// TwinCAT 3 PLC project Universalsteuerung_0663
// ProgramVersion: 3.1.4026.13
// libraries:
//   QSC_Einzelschritte, * (Q+S Control AG)
//   Tc2_MC2, * (Beckhoff Automation GmbH)
//   Tc2_Standard, * (Beckhoff Automation GmbH)
//   Tc2_SUPS, * (Beckhoff Automation GmbH)
//   Tc2_System, * (Beckhoff Automation GmbH)
//   Tc2_Utilities, * (Beckhoff Automation GmbH)
//   Tc3_EventLogger, * (Beckhoff Automation GmbH)
//   Tc3_IotBase, * (Beckhoff Automation GmbH)
//   Tc3_JsonXml, * (Beckhoff Automation GmbH)
//   Tc3_Module, * (Beckhoff Automation GmbH)
//   VisuDialogs, * (System)
//   VisuSymbols,3.5.10.0,System
// project tree:
//   DUTs/Enums/ AblaufStatus.TcDUT, AktorStatus.TcDUT, Artikeltyp.TcDUT, InitStatus.TcDUT, ResetStatus.TcDUT, StatusbarFarbe.TcDUT, StatusGreifer.TcDUT, StatusZufuehrung.TcDUT, Wartungen.TcDUT
//   DUTs/Enums/Apromace/ Antwort.TcDUT, AuftragsStatus.TcDUT, MessageArt.TcDUT
//   DUTs/Structs/EL9227_Überstromschutzklemme/ ST_BIT2.TcDUT, ST_Control.TcDUT, ST_EL9227_IN.TcDUT, ST_Status.TcDUT
//   DUTs/Structs/ ST_Ablauf_Konfig.TcDUT, ST_ArtikelParameter.TcDUT, ST_AufnahmeInfo.TcDUT, ST_EventTabelle.TcDUT, ST_Programme.TcDUT, ST_Aktor_Konfig.TcDUT, ST_QrCode.TcDUT, ST_Reihenfolge.TcDUT, ST_SchrittQueue.TcDUT, ST_Station.TcDUT, ST_Stueckzaehler.TcDUT, ST_UeberstromTabelle.TcDUT, ST_Wartung.TcDUT
//   / GlobalTextList.TcGTLO, PlcTask.TcTTO, VisualizationManager.TcVMO (not stored), VISU_TASK.TcTTO
//   GVLs/ ArtikelParam.TcGVL, Exc.TcGVL, Parameter.TcGVL
//   POUs/EventLogger/ EventLogger.TcPOU, FB_Arguments.TcPOU, FB_Event.TcPOU
//   POUs/ FB_Aktor.TcPOU, FB_Datei.TcPOU, FB_EL9227.TcPOU, FB_Handheld.TcPOU, FB_Hmi.TcPOU, FB_Output.TcPOU, FB_Schrittbetrieb.TcPOU, FB_Station01.TcPOU, FB_Stundenleistung.TcPOU, FB_Turmleuchte.TcPOU, FB_Wartung.TcPOU, FB_Zykluszeit.TcPOU, MAIN.TcPOU, Tools.TcPOU
//   POUs/Interfaces/ IF_Station.TcIO, IF_TeilBereitstellen.TcIO, IF_TeilHolen.TcIO
//   POUs/StdStationen/ FB_Station.TcPOU, FB_StationMitZuf.TcPOU, FB_StationMitZufUndVer.TcPOU
//   VISUs/ Konfig2.TcVIS, TL_Aktoren.TcTLO, Diagnose.TcVIS, EventLogger.TcVIS, TL_JaNein.TcTLO, Wartung.TcVIS, Handbetrieb.TcVIS, Konfig1.TcVIS, ImagePool.TcIPO (not stored), Zyklusbetrieb.TcVIS
// real-time tasks:
//   TASK PlcTask: cycle T#10ms, priority 20, ADS port 350
//   TASK VISU_TASK: cycle T#50000us, priority 30, ADS port 351
// I/O:
//   DEVICE Device 1 (EtherCAT), AmsNetId 10.200.30.201.2.1
//     601A1 (EK1100) [EK1100 EtherCAT Coupler (2A E-Bus)]
//       601A2 (EL9227-5500) [EL9227-5500 Overcurrent protection 24V DC, 2Ch., max. 10A (sum), adjustable, extended functionalities]
//       601A3 (EL2911) [EL2911, Potential supply terminal (10 A) with 4 Ch. Safety Inputs, TwinSAFE]
//         modules: Module 2 (FSOUT), Module 3 (DEVICEIO), Module 4 (FSLOGIC)
//       601A5 (EL9227-5500) [EL9227-5500 Overcurrent protection 24V DC, 2Ch., max. 10A (sum), adjustable, extended functionalities]
//       602A1(EL1008) [EL1008 8Ch. Dig. Input 24V, 3ms]
//       602A2 (EL2008-0015) [EL2008-0015 8Ch. Dig. Output 24V DC, 0.35A, not short-circuit proof]
//       602A4 (EL9184) [EL9184 Potential Connection, 8 x 24V, 8 x Ground]
//       (EL9011) [EL9011 End Terminal]
//     Box 15 (EP2339-0003) [EP2339-0003 16 Ch. Dig. Input/Output 24V, 0,5A, 10-Pole Plug Connector]
//     Box 16 (CTEU-EtherCAT Modular) [CTEU-EtherCAT Fieldbus modular]
//       modules: Module 1 (VAEM-L1-S-8-PT [16DO])
// variable links:
//   Universalsteuerung_0663/Universalsteuerung_0663 Instance <-> Device 1 (EtherCAT)/601A1 (EK1100)/601A2 (EL9227-5500)
//     PlcTask Inputs/MAIN.fb601A2.stKanal[1].nCurrent <-> OCP Inputs Channel 1/Current
//     PlcTask Inputs/MAIN.fb601A2.stKanal[2].nCurrent <-> OCP Inputs Channel 2/Current
//     PlcTask Inputs/MAIN.fb601A2.stKanal[1].nLoad <-> OCP Inputs Channel 1/Load
//     PlcTask Inputs/MAIN.fb601A2.stKanal[2].nLoad <-> OCP Inputs Channel 2/Load
//     PlcTask Inputs/MAIN.fb601A2.stKanal[1].nVoltageIn <-> OCP Inputs Channel 1/Voltage In
//     PlcTask Inputs/MAIN.fb601A2.stKanal[2].nVoltageIn <-> OCP Inputs Channel 2/Voltage In
//     PlcTask Inputs/MAIN.fb601A2.stKanal[1].nVoltageOut <-> OCP Inputs Channel 1/Voltage Out
//     PlcTask Inputs/MAIN.fb601A2.stKanal[2].nVoltageOut <-> OCP Inputs Channel 2/Voltage Out
//     PlcTask Inputs/MAIN.fb601A2.stKanal[1].stStatus <-> OCP Inputs Channel 1/Status
//     PlcTask Inputs/MAIN.fb601A2.stKanal[2].stStatus <-> OCP Inputs Channel 2/Status
//     PlcTask Outputs/MAIN.fb601A2.stKanal[1].stControl <-> OCP Outputs Channel 1/Control
//     PlcTask Outputs/MAIN.fb601A2.stKanal[2].stControl <-> OCP Outputs Channel 2/Control
//   Universalsteuerung_0663/Universalsteuerung_0663 Instance <-> Device 1 (EtherCAT)/601A1 (EK1100)/601A3 (EL2911)
//     PlcTask Inputs/MAIN.bE_LampeNHReset <-> StandardInputs/TwinSafeGroup1.LampeNHResetOutSPS_14
//     PlcTask Inputs/MAIN.bE_LampeNotHalt <-> StandardInputs/TwinSafeGroup1.LampeNotHaltOutSPS_88
//     PlcTask Inputs/MAIN.bE_NotHalt <-> StandardInputs/TwinSafeGroup1.NotHaltOutSPS_19
//     PlcTask Inputs/MAIN.bE_SafetyComErr <-> StandardInputs/TwinSafeGroup1.ComError_16
//     PlcTask Inputs/MAIN.bE_SafetyInRun <-> StandardInputs/TwinSafeGroup1.SafetyInRun_86
//     PlcTask Inputs/MAIN.bE_SafetyOtherErr <-> StandardInputs/TwinSafeGroup1.OtherError_17
//     PlcTask Inputs/MAIN.bE_SafetyProgStop <-> StandardInputs/TwinSafeGroup1.ProgStop_64
//     PlcTask Outputs/MAIN.bA_Hauptventil <-> StandardOutputs/TwinSafeGroup1.HauptventilSPS_48
//     PlcTask Outputs/MAIN.bA_SafetyReset <-> StandardOutputs/TwinSafeGroup1.ErrorAcknowledgement_1
//     PlcTask Outputs/MAIN.bA_SafetyRun <-> StandardOutputs/TwinSafeGroup1.Run_47
//   Universalsteuerung_0663/Universalsteuerung_0663 Instance <-> Device 1 (EtherCAT)/601A1 (EK1100)/601A5 (EL9227-5500)
//     PlcTask Inputs/MAIN.fb601A5.stKanal[1].nCurrent <-> OCP Inputs Channel 1/Current
//     PlcTask Inputs/MAIN.fb601A5.stKanal[2].nCurrent <-> OCP Inputs Channel 2/Current
//     PlcTask Inputs/MAIN.fb601A5.stKanal[1].nLoad <-> OCP Inputs Channel 1/Load
//     PlcTask Inputs/MAIN.fb601A5.stKanal[2].nLoad <-> OCP Inputs Channel 2/Load
//     PlcTask Inputs/MAIN.fb601A5.stKanal[1].nVoltageIn <-> OCP Inputs Channel 1/Voltage In
//     PlcTask Inputs/MAIN.fb601A5.stKanal[2].nVoltageIn <-> OCP Inputs Channel 2/Voltage In
//     PlcTask Inputs/MAIN.fb601A5.stKanal[1].nVoltageOut <-> OCP Inputs Channel 1/Voltage Out
//     PlcTask Inputs/MAIN.fb601A5.stKanal[2].nVoltageOut <-> OCP Inputs Channel 2/Voltage Out
//     PlcTask Inputs/MAIN.fb601A5.stKanal[1].stStatus <-> OCP Inputs Channel 1/Status
//     PlcTask Inputs/MAIN.fb601A5.stKanal[2].stStatus <-> OCP Inputs Channel 2/Status
//     PlcTask Outputs/MAIN.fb601A5.stKanal[1].stControl <-> OCP Outputs Channel 1/Control
//     PlcTask Outputs/MAIN.fb601A5.stKanal[2].stControl <-> OCP Outputs Channel 2/Control
//   Universalsteuerung_0663/Universalsteuerung_0663 Instance <-> Device 1 (EtherCAT)/601A1 (EK1100)/602A1(EL1008)
//     PlcTask Inputs/MAIN.bE_LuftdruckIO <-> Channel 5/Input
//     PlcTask Inputs/MAIN.bE_Taste_Schritt <-> Channel 4/Input
//     PlcTask Inputs/MAIN.bE_Taste_Start <-> Channel 1/Input
//     PlcTask Inputs/MAIN.bE_Taste_Stoerung <-> Channel 3/Input
//     PlcTask Inputs/MAIN.bE_Taste_Stop <-> Channel 2/Input
//   Universalsteuerung_0663/Universalsteuerung_0663 Instance <-> Device 1 (EtherCAT)/601A1 (EK1100)/602A2 (EL2008-0015)
//     PlcTask Outputs/MAIN.bA_Lampe_NHReset <-> Channel 4/Output
//     PlcTask Outputs/MAIN.bA_Lampe_NotHalt <-> Channel 5/Output
//     PlcTask Outputs/MAIN.bA_Lampe_Schritt <-> Channel 6/Output
//     PlcTask Outputs/MAIN.bA_Lampe_Start <-> Channel 1/Output
//     PlcTask Outputs/MAIN.bA_Lampe_Stoerung <-> Channel 3/Output
//     PlcTask Outputs/MAIN.bA_Lampe_Stop <-> Channel 2/Output
//   Universalsteuerung_0663/Universalsteuerung_0663 Instance <-> Device 1 (EtherCAT)/Box 15 (EP2339-0003)
//     PlcTask Inputs/MAIN.bE_Fussschalter <-> DI Inputs Channel 2/Input 1
//     PlcTask Inputs/MAIN.fbSt1.bE_Sensor[{1..8}] <-> DI Inputs Channel 1/Input {1..8}  (8 links)
//     PlcTask Outputs/MAIN.fbSt1.bA_extGeraetStart <-> DO Outputs Channel 2/Output 2
//   Universalsteuerung_0663/Universalsteuerung_0663 Instance <-> Device 1 (EtherCAT)/Box 16 (CTEU-EtherCAT Modular)
//     PlcTask Outputs/MAIN.fbSt1.fbAktor[1].bA_arbeitsPos <-> Module 1 (VAEM-L1-S-8-PT [16DO])/Outputs/C1 Output[0]
//     PlcTask Outputs/MAIN.fbSt1.fbAktor[2].bA_arbeitsPos <-> Module 1 (VAEM-L1-S-8-PT [16DO])/Outputs/C1 Output[2]
//     PlcTask Outputs/MAIN.fbSt1.fbAktor[3].bA_arbeitsPos <-> Module 1 (VAEM-L1-S-8-PT [16DO])/Outputs/C1 Output[4]
//     PlcTask Outputs/MAIN.fbSt1.fbAktor[4].bA_arbeitsPos <-> Module 1 (VAEM-L1-S-8-PT [16DO])/Outputs/C1 Output[6]
//     PlcTask Outputs/MAIN.fbSt1.fbAktor[5].bA_arbeitsPos <-> Module 1 (VAEM-L1-S-8-PT [16DO])/Outputs/C2 Output[0]
//     PlcTask Outputs/MAIN.fbSt1.fbAktor[6].bA_arbeitsPos <-> Module 1 (VAEM-L1-S-8-PT [16DO])/Outputs/C2 Output[2]

CONFIGURATION Universalsteuerung_0663
    RESOURCE PLC ON TwinCAT3
        TASK PlcTask(INTERVAL := T#10ms, PRIORITY := 20);
        TASK VISU_TASK(INTERVAL := T#50000us, PRIORITY := 30);
        PROGRAM MAIN WITH PlcTask : MAIN;
        PROGRAM VisuElems_Visu_Prg WITH VISU_TASK : VisuElems.Visu_Prg;
    END_RESOURCE
END_CONFIGURATION

// ---- DUTs/Enums/AblaufStatus.TcDUT
{attribute 'qualified_only'}
//{attribute 'strict'}
{attribute 'to_string'}
TYPE AblaufStatus :
(
//	default				:= 0,
//	bereit				:= 1,
//	error				:= 2,
//	produziert			:= 3,
//	fertig				:= 5,
//	popUp				:= 6,
	
//	aktor01Vor			:= 10,
//	aktor01Zurueck		:= 11,
//	aktor02Vor			:= 20,
//	aktor02Zurueck		:= 21,
//	aktor03Vor			:= 30,
//	aktor03Zurueck		:= 31,
//	aktor04Vor			:= 40,
//	aktor04Zurueck		:= 41,
//	aktor05Vor			:= 50,
//	aktor05Zurueck		:= 51,
//	aktor06Vor			:= 60,
//	aktor06Zurueck		:= 61,
	
//	teilAnwesend		:= 80,
//	extGeraetBereit		:= 81,
//	extGeraetStart		:= 82,
//	warten				:= 90,
	
//	nameUeberpruefen 	:= 200,
//	freierPlatzsuchen 	:= 201,
//	programmSpeichern 	:= 202,
//	programmAnzeigen	:= 203,
//	programmLoeschen	:= 204

	default				:= 0,
	aktor01Vor			:= 1,
	aktor01Zurueck		:= 2,
	aktor02Vor			:= 3,
	aktor02Zurueck		:= 4,
	aktor03Vor			:= 5,
	aktor03Zurueck		:= 6,
	aktor04Vor			:= 7,
	aktor04Zurueck		:= 8,
	aktor05Vor			:= 9,
	aktor05Zurueck		:= 10,
	aktor06Vor			:= 11,
	aktor06Zurueck		:= 12,
	teilAnwesend		:= 13,
	extGeraetBereit		:= 14,
	extGeraetStart		:= 15,
	extGeraetFertig		:= 16,
	warten				:= 17,
	schritt				:= 18,
	
	bereit				:= 30,
	error				:= 31,
	produziert			:= 32,
	fertig				:= 33,
	popUp				:= 34,
	naechsterSchritt	:= 35,
	
	nameUeberpruefen 	:= 200,
	freierPlatzsuchen 	:= 201,
	programmSpeichern 	:= 202,
	programmAnzeigen	:= 203,
	programmLoeschen	:= 204,
	
	oeffnen				:= 300,
	wartenOffen			:= 301,
	schreiben			:= 302,
	wartenGeschrieben	:= 303,
	schliessen			:= 304,
	wartenGeschlossen	:= 305
	
	
	

	
);
END_TYPE

// ---- DUTs/Enums/AktorStatus.TcDUT
{attribute 'qualified_only'}
{attribute 'strict'}
{attribute 'to_string'}
TYPE AktorStatus :
(
	default := 0,
	inRP,
	inAP,
	
	zuRP,
	zuAP
);
END_TYPE

// ---- DUTs/Enums/Apromace/Antwort.TcDUT
{attribute 'qualified_only'}
{attribute 'strict'}
TYPE Antwort :
(
	pending,	//wartet auf Antwort
	timeout,
	ok,
	error,
	ignored,	//Ignore flag aktiviert
	expired		//Quittiert nach Error
);
END_TYPE

// ---- DUTs/Enums/Apromace/AuftragsStatus.TcDUT
{attribute 'qualified_only'}
{attribute 'strict'}
TYPE AuftragsStatus :
(
	scan,
	start,
	end,
	vorwahl
);
END_TYPE

// ---- DUTs/Enums/Apromace/MessageArt.TcDUT
{attribute 'qualified_only'}
{attribute 'strict'}
{attribute 'to_string'}
TYPE MessageArt :
(
	status,
	auftrag,
	daten,
	parameter
);
END_TYPE

// ---- DUTs/Enums/Artikeltyp.TcDUT
{attribute 'qualified_only'}
{attribute 'strict'}
{attribute 'to_string'}
TYPE Artikeltyp :
(
	default 				:= 0,
	br51,
	br84
);
END_TYPE

// ---- DUTs/Enums/InitStatus.TcDUT
{attribute 'qualified_only'}
{attribute 'strict'}
{attribute 'to_string'}
TYPE InitStatus :
(
	default := 0,
	bereit,
	steuerungEin,
	safety,
	resetSafety,
	luftdruck,
	fertig,
	stationen,
	aktor1,
	aktor2,
	aktor3,
	aktor4,
	aktor5,
	aktor6
);
END_TYPE

// ---- DUTs/Enums/ResetStatus.TcDUT
{attribute 'qualified_only'}
{attribute 'strict'}
{attribute 'to_string'}
TYPE ResetStatus :
(
	default := 0,
	bereit,
	ablaufAbbrechen,
	ausschalten,
	fertig,
	aktoren,
	kommunikationAbgebrochen
);
END_TYPE

// ---- DUTs/Enums/StatusbarFarbe.TcDUT
{attribute 'qualified_only'}
TYPE StatusbarFarbe :
(
	default := 0,
	rot :=1,
	orange := 2,
	gruen := 3,
	blau := 4
);
END_TYPE

// ---- DUTs/Enums/StatusGreifer.TcDUT
{attribute 'qualified_only'}
{attribute 'strict'}
{attribute 'to_string'}
TYPE StatusGreifer :
(
	default := 0,
	keinTeil,
	teilHolen,
	teilGeholt,
	teilEinlegen,
	teilEntnehmen,
	teilEntnommen,
	teilAblegen,
	teilAbgelegt,
	teilGegriffen,
	teilGegriffenDrehen,
	lagerplatte,
	lagerplatteMitFeder,
	ausschuss,
	blockiert
);
END_TYPE

// ---- DUTs/Enums/StatusZufuehrung.TcDUT
{attribute 'qualified_only'}
{attribute 'strict'}
{attribute 'to_string'}
TYPE StatusZufuehrung :
(
	default := 0,
	bereit,						//Entstören Stau
	keinTeil,					// Ablauf
	teilHolen,					// Ablauf
	teilVereinzelt,				// Ablauf
	teilEntnommen, 				// Ablauf
	fertig						// Ablauf

);
END_TYPE

// ---- DUTs/Enums/Wartungen.TcDUT
{attribute 'qualified_only'}
{attribute 'strict'}
TYPE Wartungen :
(
	nothaltAustauschen			:= 1,
	zweihandSchalterAustauschen	:= 2
);
END_TYPE

// ---- DUTs/Structs/EL9227_Überstromschutzklemme/ST_BIT2.TcDUT
TYPE ST_BIT2 :
STRUCT
	a:BIT;
	b:BIT;
END_STRUCT
END_TYPE

// ---- DUTs/Structs/EL9227_Überstromschutzklemme/ST_Control.TcDUT
TYPE ST_Control :
STRUCT
	bReset:		BOOL;
	bSwitch:	BOOL;
END_STRUCT
END_TYPE

// ---- DUTs/Structs/EL9227_Überstromschutzklemme/ST_EL9227_IN.TcDUT
TYPE ST_EL9227_IN :
STRUCT
	stStatus	AT%I*:	ST_Status;
	nLoad		AT%I*:	UINT;
	nCurrent	AT%I*:	UINT;
	nVoltageIn	AT%I*:	UINT;
	nVoltageOut	AT%I*:	UINT;
	stControl	AT%Q*:	ST_Control;
END_STRUCT
END_TYPE

// ---- DUTs/Structs/EL9227_Überstromschutzklemme/ST_Status.TcDUT
TYPE ST_Status :
STRUCT
	bEnabled:				BIT;
	bTripped:				BIT;
	bShortCircuit:			BIT;
	bOverload:				BIT;
	bHardwareProtection:	BIT;
	bOvervoltage:			BIT;
	bUndervoltage:			BIT;
	bCurrentLevelWarning:	BIT;
	bCoolDownLock:			BIT;
	bDisabledBySwitch:		BIT;
	bDisabledByDI:			BIT;
	bDisabledByOutput:		BIT;
	bDiag:					BIT;
	bTxPDOState:			BIT;
	bInputCycleCounter:		ST_BIT2;
	bStateDeviceSwitch:		BIT;
	bStateDigitalInput:		BIT;
	bError:					BIT;
	bStateReset:			BIT;
	bStateSwitch:			BIT;
END_STRUCT
END_TYPE

// ---- DUTs/Structs/ST_Ablauf_Konfig.TcDUT
TYPE ST_Ablauf_Konfig :
STRUCT
	nNummer:				UINT;
	eAblaufStatus:			AblaufStatus;
END_STRUCT
END_TYPE

// ---- DUTs/Structs/ST_ArtikelParameter.TcDUT
TYPE ST_ArtikelParameter :
STRUCT
	//Prüfling
	sArtikel:						STRING; // Vorwahl
	sFullArtikelNr:					STRING;
	sBezeichung:					STRING; // Vorwahl
	sAuftragsNr:					STRING;
	eTyp:							Artikeltyp;

	nAuftragsMenge:					UINT;
	
	fMinLaengeBolzen:				REAL;
	fMaxLaengeBolzen:				REAL;
	
	fMinLaengeGesamt:				REAL;
	fMaxLaengeGesamt:				REAL;
END_STRUCT
END_TYPE

// ---- DUTs/Structs/ST_AufnahmeInfo.TcDUT
TYPE ST_AufnahmeInfo :
STRUCT
	//Arbeitsschritte
	
	//Infos
	bFertig:					BOOL;		//Teil fertig oder Ausschuss (kann entnommen werden)
	bAusschuss:					BOOL;
	
	fLaengeBolzen1:				REAL;
	fLaengeBolzen2:				REAL;
	fLaengeGesamt:				REAL;
	
	//nFehlerCodeMontage:			LWORD;
	(*Fehlercodes:
	Bit|Grund
	0	Lagerplatte Pos 1 nicht in Toleranz
	1	Lagerplatte Pos 2 nicht in Toleranz
	2	Lagerplatte Pos 3 nicht in Toleranz
	3	Lagerplatte Pos 1 erkannt obwohl keine Bestückt werden sollte
	4	Lagerplatte Pos 2 erkannt obwohl keine Bestückt werden sollte
	5	Lagerplatte Pos 3 erkannt obwohl keine Bestückt werden sollte
	*)
	
	//Artikelparameter
	stArtParam:					ST_ArtikelParameter;
	
END_STRUCT
END_TYPE

// ---- DUTs/Structs/ST_EventTabelle.TcDUT
TYPE ST_EventTabelle :
STRUCT
	sSeverity:			STRING;
	sStatus:			STRING;
	sTimestamp:			STRING;
	sText:				STRING(255);
	nEventId:			INT;
	bPinned:			BOOL;
END_STRUCT
END_TYPE

// ---- DUTs/Structs/ST_Programme.TcDUT
TYPE ST_Programme :
STRUCT
	nNr:			INT;
	sName:			STRING;
	aAktorBew:		ARRAY [1..Parameter.cAnzSchritte] OF ST_Ablauf_Konfig;
	aAktorKonfig:	ARRAY [1..Parameter.cAnzAktoren] OF ST_Aktor_Konfig;
	nTeilAnw:			INT;
	nFussschalterAktiv: INT;			// 0 = Ja / 1 = Nein
END_STRUCT
END_TYPE

// ---- DUTs/Structs/ST_Aktor_Konfig.TcDUT
TYPE ST_Aktor_Konfig :
STRUCT
	//eTyp:					Aktortyp;					braucht es dies?
	//nNummer:				UINT;						ist neu in ST_Ablauf_Konfig
	//eAblaufStatus:		AblaufStatus;				ist neu in ST_Ablauf_Konfig
	//bSensRuhePos:			BOOL;						neu als INT, Dropdown im HMI
	//bSensArbeitsPos:		BOOL;						neu als INT, Dropdown im HMI
	nSensRuhePos:			INT;
	nSensArbeitsPos:		INT;
	nFahrZeit:				UINT;
	tFahrZeit:				TIME;
	nHalteZeit:				UINT;
	tHalteZeit:				TIME;
	bReversierBetrieb:		BOOL;
	
END_STRUCT
END_TYPE

// ---- DUTs/Structs/ST_QrCode.TcDUT
TYPE ST_QrCode :
STRUCT
	sAuftrag:			STRING;
	sArtikel:			STRING;
	sAuftragsmenge:		STRING;
	sEndTermin:			STRING;
	
	bGueltig:			BOOL;
END_STRUCT
END_TYPE

// ---- DUTs/Structs/ST_Reihenfolge.TcDUT
TYPE ST_Reihenfolge :
STRUCT
	eAblauf: AblaufStatus;
	eLetzterStatus: AblaufStatus;
	tFahrzeit: TIME;
	tHaltezeit: TIME;
END_STRUCT
END_TYPE

// ---- DUTs/Structs/ST_SchrittQueue.TcDUT
TYPE ST_SchrittQueue :
STRUCT
	fbAktor:				REFERENCE TO FB_Aktor;
	fbOutput:				REFERENCE TO FB_Output;
	bInPos:					BOOL;						//Ob Sollposition erreicht wurde
	bGesetzt:				BOOL;						//Information ob ausgang gesetzt oder zurueckgesetzt wurde (arbeitsPos -> gesetzt)
	bStatuswechsel:			BOOL;						//True wenn nach diesem Eintrag der Status des Ablaufs gewechselt hat
END_STRUCT
END_TYPE

// ---- DUTs/Structs/ST_Station.TcDUT
TYPE ST_Station :
STRUCT
	bRstStop:			BOOL;		//Schreibt Station
	bInit:				BOOL;		//Schreibt Main
	bInitBeendet:		BOOL;		//Schreibt Station
	bReset:				BOOL;
	bStoerung:			BOOL;		//Anlage blockiert
	bWarnung:			BOOL;		//Könnte verzögerungen verursachen
	nStationsNr:		INT;
	
	bZyklusFertig:		BOOL;
	sStatus:			STRING;
END_STRUCT
END_TYPE

// ---- DUTs/Structs/ST_Stueckzaehler.TcDUT
TYPE ST_Stueckzaehler :
STRUCT
	nGutteileTag:		UINT;
	nGutteileGesamt:	UDINT;
	nGutteileAuftrag:	UINT;
	
	nAusschussTag:		UINT;
	nAusschussGesamt:	UDINT;
	nAusschussAuftrag:	UINT;
	
	nAuftragszaehler:	UINT;
	nGesamt:			UDINT;
	
END_STRUCT
END_TYPE

// ---- DUTs/Structs/ST_UeberstromTabelle.TcDUT
TYPE ST_UeberstromTabelle :
STRUCT
	// Status
	sKlemme:				STRING;
	sKanal:					STRING;
	sLoad:					STRING;
	sCurrent:				STRING;
	sVoltageIn:				STRING;
	sVoltageOut:			STRING;
	sEnabled:				STRING;
	sTripped:				STRING;
	sShortCircuit:			STRING;
	sOverload:				STRING;
	sHardwareProtection:	STRING;
	sOvervoltage:			STRING;
	sUndervoltage:			STRING;
	sCurrentLevelWarning:	STRING;
	sCoolDownLock:			STRING;
	sDisabledBySwitch:		STRING;
	sDisabledByDI:			STRING;
	sDisabledByOutput:		STRING;
	
	
	
	
	
END_STRUCT
END_TYPE

// ---- DUTs/Structs/ST_Wartung.TcDUT
TYPE ST_Wartung :
STRUCT
	sBezeichnung:		STRING;
	sPerson:			STRING;			//Wer die Wartung durchführen darf

	nZyklenBisWartung:	LINT;			//nach wie vielen Zyklen die wartung durchgeführt werden muss
	fZeitBisWartung:	REAL;			//nach welcher Zeit die wartung durchgeführt werden muss
	
	nZyklenSeitWartung:	LINT;
	fZeitSeitWartung:	LREAL;
	bAnstehend:			BOOL;
	
	sVerbleibendeZeit:	STRING;
	sVerbleibendeZyklen:STRING;
	
	sZyklenBisWartung:	STRING;
	sZeitBisWartung:	STRING;

	bBtnReset:			BOOL;
END_STRUCT
END_TYPE

// ---- GVLs/ArtikelParam.TcGVL
{attribute 'qualified_only'}
VAR_GLOBAL
	akt:					ST_ArtikelParameter;
END_VAR

// ---- GVLs/Exc.TcGVL
{attribute 'qualified_only'}
VAR_GLOBAL
	nCheckBounds              : INT;
    nCheckBounds_OutOfBoundsUpper  : INT;
	nCheckBounds_OutOfBoundsLower  : INT;
    myException               : __SYSTEM.ExceptionCode;
END_VAR

// ---- GVLs/Parameter.TcGVL
{attribute 'qualified_only'}
VAR_GLOBAL	
	
END_VAR

VAR_GLOBAL CONSTANT
	
	//Allegemein
	cAnzStationen:				INT := 1;
	cAnzAktoren:				INT := 6;
	cAnzSchritte:				INT := 12;
	cAnzEvents:					INT := 300;
	cAnzLoggedEvents:			INT := 100;
	cAktRateStundenLeistung:	INT := 30;
	
	cGroesseSchrittQueue:		INT := 100;
	
	fZyklusZeitTask:			REAL := 10;	//ms
	cMaschinenInfo:				STRING := '0660.0000 / Zweihandausloesung';
	

	//Aktoren
	cZylZeit:					TIME := T#700MS;
	cZylUeberwachung:			TIME := T#1S;
	cZylUeberwachung2s:			TIME := T#2S;
	cZylUeberwachung3s:			TIME := T#3S;
	cZangeUeberwachung:			TIME := T#300MS;
	cDreherUeberwachung:		TIME := T#1S;
	cZangeZeit:					TIME := T#100MS;
	cZangeZeit2:				TIME := T#200MS;
	cZangeZeit3:				TIME := T#300MS;
	cDreherZeit:				TIME := T#200MS;
	cBlockierungZeit:			TIME := T#100MS;
	cZeitZwischenanschlag:		TIME := T#100MS;
		
	//Station 1
	cPresseFehlerZeit:			TIME := T#5000MS;

	//MQTT 
	cJsonLenApromace:			UINT := 5000;
	
	// Programmhandling
	cMaxProgramme:				INT := 100;
	
	
	
	//Wartungen		
	cAnzWartungen:				INT := 1;	
	cMaxZyklNotHalt:			DINT := 2500;		// Gem. SISTEMA 2500 Zyklen		
	aWartungenConfig:			ARRAY[1..Parameter.cAnzWartungen] OF ST_Wartung :=
								//Liste der Wartungen 
								[	
								(	sBezeichnung		:= 'Not-Halt austauschen',
									sPerson				:= 'Betriebsmechaniker',
									nZyklenBisWartung	:= 100000,
									fZeitBisWartung 	:= 0)];			//in h
									
	//CSV
	sPfad:						STRING := '\Hard Disk2\';
	cAnzCSVStrings:				INT := 1000;
									
END_VAR

VAR_GLOBAL PERSISTENT
	nAnzAusschussBisStoerung:	INT;

END_VAR

// ---- POUs/Interfaces/IF_Station.TcIO
INTERFACE IF_Station

METHOD bearbeitenAnfordern
VAR_INPUT
	nAufnahme:		INT;
END_VAR
END_METHOD

METHOD init : BOOL
VAR_INPUT
END_VAR
END_METHOD

METHOD reset : BOOL
VAR_INPUT
END_VAR
END_METHOD

METHOD teilBearbeiten : BOOL
VAR_INPUT
END_VAR
END_METHOD

END_INTERFACE

// ---- POUs/Interfaces/IF_TeilBereitstellen.TcIO
INTERFACE IF_TeilBereitstellen

METHOD holenAnfordern
VAR_INPUT
END_VAR
END_METHOD

METHOD teilBereitstellen : BOOL
VAR_INPUT
END_VAR
END_METHOD

END_INTERFACE

// ---- POUs/Interfaces/IF_TeilHolen.TcIO
INTERFACE IF_TeilHolen

METHOD holenAnfordern
VAR_INPUT
END_VAR
END_METHOD

METHOD teilHolen : BOOL
VAR_INPUT
END_VAR
END_METHOD

END_INTERFACE

// ---- POUs/MAIN.TcPOU
PROGRAM MAIN
VAR_INPUT	
	//Aktoren
	bPosNachHbNio:			BOOL;
	
	//FBs
	HMI:					FB_Hmi;	
	fbTurmleuchte:			FB_Turmleuchte;
	
	nAusschussZaehler:		INT;
	bLampeStoerung:			BOOL;
	
	stAufnahmeInfo:			ST_AufnahmeInfo;
	bProduzieren:			BOOL;
	bAuftragLaeuft:			BOOL;
	bZyklusZeitMessStart:	BOOL;
	bWritePersistentMan:	BOOL;
	fbSt1:					FB_Station01;	

END_VAR
VAR
	//Safety
	bE_NotHalt				AT%I*:	BOOL;
	bA_SafetyReset			AT%Q*:	BOOL;
	bA_SafetyRun			AT%Q*:	BOOL := TRUE;   
	bA_TasteNHReset			AT%Q*:	BOOL;
	bA_Hauptventil			AT%Q*:	BOOL;
    
	bE_SafetyComErr			AT%I*:	BOOL;
	bE_SafetyOtherErr		AT%I*:	BOOL;
	bE_SafetyProgStop		AT%I*:	BOOL;
	bE_busVerbVerloren 		AT%I*:	BOOL;		//Busverbindung verloren (WC STATE Klemme 1)
	bE_SafetyInRun			AT%I*:	BOOL;
	bE_TasteNHReset			AT%I*:	BOOL;
	bE_LampeNHReset			AT%I*:	BOOL;
	bE_LampeNotHalt			AT%I*:	BOOL;
	
	bE_Handbetrieb:					BOOL;	
	
	//Tasten
	bE_Taste_Start			AT%I*:	BOOL;
	bE_Fussschalter			AT%I*:	BOOL;
	bE_Taste_Stop			AT%I*:	BOOL;
	bE_Taste_Stoerung		AT%I*:	BOOL;
	bE_Taste_Schritt		AT%I*:	BOOL;
	
	//Lampen
	bA_Lampe_Start			AT%Q*:	BOOL;
	bA_Lampe_Stop			AT%Q*:	BOOL;
	bA_Lampe_Stoerung		AT%Q*:	BOOL;
	bA_Lampe_NHReset		AT%Q*:	BOOL;
	bA_Lampe_NotHalt		AT%Q*:	BOOL;
	bA_Lampe_Schritt		AT%Q*:	BOOL;
	
	//Tasten Flanken
	fbStartFlanke:			R_TRIG;
	fbStopFlanke:			R_TRIG;
	fbStoerungFlanke:		R_TRIG;

	
	//Sonstige Inputs
	bE_LuftdruckIO			AT%I*:	BOOL;	
	
	//Init
	eInitStatus:			InitStatus := InitStatus.bereit;
	
	//Stationen
	aStationInfo:			ST_Station;
	bInitStNr:				BOOL := TRUE;
	
	//MQTT
	//fbMqttApromace:			FB_MqttApromace;
	nStoerungsgrund:		INT;
	
	//Sonstiges
	i:						INT;
	sMqttStatus:			STRING;
	sMqttVorher:			STRING;
	fbSystemZeit:			NT_GetTime;
	
	eStartAblauf1:			AblaufStatus := AblaufStatus.bereit;
	//fbStartMessage:			FB_Message;
	
	sFehlerText:			STRING(255);	
	bStoerung:				BOOL;
	bWarnung:				BOOL;
	
	bLampenTest:			BOOL;
	
	bInitBeendet:			BOOL;
	
	SafetyAck: 				INT:=1;
	fbErrTP: 				TP;
	
	
	bZyklusGestartet:		BOOL;
	bStopNachZyklus:		BOOL;
		
	//Stationen
	//fbSt1:					FB_Station01;	

	
	//Sonstige FBs	
	fbBlinkZeit:			TON;
	fbWritePersistentData: 	WritePersistentData;
	fbWritePersistent:		R_TRIG;
	fbTofLuft:				TOF;
	fbHandheld:				FB_Handheld;
	fbUsv:					FB_S_UPS_CB3011;
	
	
	
	//IPC Daten
	sSrcNetId: 				T_AmsNetId;						//Lokale NetId
	
	// Zykluszeit
	fbZyklusZeitGesamt:		FB_Zykluszeit;
	
	//FB's Überstromschutzklemmen (ACHTUNG: Nicht die neuste Version)
	fb601A2: 				FB_EL9227(	nErrorId:= 260, 
										sBezeichnung:= '601A2');		
	fb601A5: 				FB_EL9227(	nErrorId:= 260, 
										sBezeichnung:= '601A5');							
	
	//Stundenleistung
	fSummeZyklus:			REAL;
	fStundenLeistung:		REAL;
	idx1:					INT := 1;
	idx2:					INT;
	fbStundenLeistungFlanke:R_TRIG;	
	fbStundenleistung:		FB_Stundenleistung;
	
	bProgStop:				BOOL;
	
	fbStatusPunkteZeit:		TON;
	sStatus:				STRING(255);
	nPunkte:				INT;
	
	sText:					STRING(255);	
	
	
	CLK: INT;
	fbWartung:				FB_Wartung;
END_VAR


VAR_INPUT PERSISTENT
	sAuftragVorher:			STRING;
	nMonatVorher:			WORD;
	nTagVorher:				WORD;
	stStueckzaehler:		ST_Stueckzaehler;
	fBetriebsstunden:		LREAL;
END_VAR

// Not-Halt von allen Stationen zusammenfassen



bA_TasteNHReset := bE_TasteNHReset;
bProgStop := bPosNachHbNio;

IF			bE_SafetyProgStop THEN
	bProgStop := TRUE;
END_IF
				
IF			bPosNachHbNio THEN
	bLampeStoerung := TRUE;
END_IF
bPosNachHbNio := FALSE;					//muss unter der verwendung sein, dass alle aktoren im Zyklus überschreiben können

//***********************************************************************************************
//Init StationsNr
IF			bInitStNr THEN
	bInitStNr := FALSE;
	FOR i := 0 TO Parameter.cAnzStationen DO
		aStationInfo.nStationsNr := i;
	END_FOR
END_IF

//***********************************************************************************************
//Stationen
fbSt1(	ifStation := fbSt1,
		stStationInfo := aStationInfo);


//MQTT
//fbMqttApromace(	sAnlagename:= 'DIV_Universalsteuerung_0661.0000-01',
//				sWerk:= 'EHQ');

//***********************************************************************************************
//Sontige FBs und PRGs
fbStartFlanke(CLK := bE_Taste_Start OR bE_Fussschalter);
fbStopFlanke(CLK := NOT bE_Taste_Stop);
fbStoerungFlanke(CLK := bE_Taste_Stoerung);





EventLogger();
HMI();
Lampen();

fbSystemZeit(	NETID := sSrcNetId,
				START := NOT fbSystemZeit.START);

// Persistente Daten schreiben über Button "bWritePersistentMan" oder über bE_BusVerbVerloren	
fbWritePersistent(CLK := bWritePersistentMan);			
fbWritePersistentData.START :=	fbWritePersistent.Q;
fbWritePersistentData(NETID:='', PORT:=851, TMOUT:=T#1S);
IF			fbWritePersistentData.BUSY THEN
	MAIN.bWritePersistentMan := FALSE;
END_IF


fbUsv(	ePersistentMode := SPDM_2PASS,
		eUpsMode :=  eSUPS_WrPersistData_Shutdown,
		sNetID := '',
		iPLCPort := 851,
		tTimeout := DEFAULT_ADS_TIMEOUT,
		tRecoverTime := T#10S);



//***********************************************************************************************
//Init
init();

//***********************************************************************************************
//Reset
IF			(bInitBeendet
	OR		(eInitStatus <> InitStatus.bereit))
	AND NOT bE_NotHalt THEN
	bProduzieren := FALSE;
	bStopNachZyklus := FALSE;
	bZyklusGestartet := FALSE;	
	bInitBeendet := FALSE;
	eInitStatus := InitStatus.bereit;
	bA_Hauptventil := FALSE;
	
	aStationInfo.bInitBeendet := FALSE;
	aStationInfo.bReset := TRUE;

END_IF

//Start Ablauf
CASE eStartAblauf1 OF
	
	//***********************************************************************************************	
	AblaufStatus.bereit:		
		IF			(fbStartFlanke.Q
			OR		 MAIN.HMI.ProgrammTemp.nFussschalterAktiv = 0)
			AND		fbst1.bNotHaltTestIO
			AND		bInitBeendet
			AND		MAIN.HMI.bProgrammgeladen
			//AND		HMI.bAuftragGeladen
			AND  	aStationInfo.bZyklusFertig
			AND NOT bE_Handbetrieb
			AND NOT	bProgStop
			AND		bE_LuftdruckIO
			AND NOT bProduzieren THEN
				fbSt1.bearbeitenAnfordern(1);
				eStartAblauf1 := AblaufStatus.produziert;
				bZyklusZeitMessStart := FALSE;
		END_IF

	//***********************************************************************************************	
	AblaufStatus.produziert:
		bZyklusZeitMessStart := TRUE;
		IF		 aStationInfo.bZyklusFertig THEN
			eStartAblauf1 := AblaufStatus.bereit;
			
		END_IF
END_CASE



//*****************************************************************
//Start Fehlermeldungen
IF			fbStartFlanke.Q
	AND 	bE_SafetyProgStop THEN
	EventLogger.aErrorLog[230].Send(0);
END_IF
//*****************************************************************
IF			fbStartFlanke.Q
	AND 	bPosNachHbNio THEN
	EventLogger.aErrorLog[231].Send(0);
END_IF
//*****************************************************************
IF			fbStartFlanke.Q
	AND 	bE_Handbetrieb THEN
	EventLogger.aErrorLog[232].Send(0);
END_IF
//*****************************************************************	
IF			fbStartFlanke.Q
	AND NOT bInitBeendet THEN
	EventLogger.aErrorLog[233].Send(0);
END_IF
//*****************************************************************
IF			fbStartFlanke.Q
	AND NOT HMI.bAuftragGeladen THEN
	EventLogger.aErrorLog[234].Send(0);
END_IF
//*****************************************************************
IF			fbStartFlanke.Q
	AND 	(nAusschussZaehler >= Parameter.nAnzAusschussBisStoerung) THEN
	EventLogger.aErrorLog[235].Send(0);
END_IF

//***********************************************************************************************
//Produktion läuft
IF		NOT aStationInfo.bZyklusFertig THEN
	bProduzieren := TRUE;
END_IF


IF		NOT aStationInfo.bZyklusFertig
	AND 	bInitBeendet THEN
	bZyklusGestartet := TRUE;
END_IF


//***********************************************************************************************
//Zähler zurücksetzen
IF		 	(nTagVorher <> fbSystemZeit.TIMESTR.wDay 
	OR 	  	nMonatVorher <> fbSystemZeit.TIMESTR.wMonth)
	AND		fbSystemZeit.TIMESTR.wMonth > 0 THEN		//Damit der fbSystemzeit sicher ausgeführt wurde
	stStueckzaehler.nGutteileTag := 0;
	stStueckzaehler.nAusschussTag := 0;
	nTagVorher := fbSystemZeit.TIMESTR.wDay;
	nMonatVorher := fbSystemZeit.TIMESTR.wMonth;
END_IF

//***********************************************************************************************
//Betriebsstunden
fBetriebsstunden := fBetriebsstunden + (Parameter.fZyklusZeitTask/3600000);

//Zykluszeiten	

IF			bInitBeendet THEN	
	fbZyklusZeitGesamt(	bStart			:= 		bZyklusZeitMessStart,
						fZyklusZeitTask	:= Parameter.fZyklusZeitTask);
END_IF


fbStundenLeistungFlanke(CLK :=  aStationInfo.bZyklusFertig);

//Stundenleistung	
fbStundenleistung(fZyklusZeitTask := Parameter.fZyklusZeitTask,
					bProduzieren := bProduzieren,
					nStueckZaehlerAnlage := stStueckzaehler.nGutteileGesamt,
					bInitBeendet := bInitBeendet,
					fStundenLeistung => fStundenLeistung);
					
//***********************************************************************************************
// Lampensäule Gruen
IF 		NOT bInitBeendet THEN
	fbTurmleuchte.warnung();
ELSIF		NOT Main.bProgStop 
		AND		bProduzieren THEN
	fbTurmleuchte.betrieb();
END_IF

//***********************************************************************************************
//Störungen


// Luftdruck n.i.O Meldung
fbTofLuft(IN:=bE_LuftdruckIO, PT:= T#500MS);

IF		NOT	fbTofLuft.Q 
	AND 	bInitBeendet
	AND	NOT	EventLogger.aAlarm[257].bRaised THEN
	EventLogger.aAlarm[257].Raise(0);
	
ELSIF		bE_LuftdruckIO
	AND		EventLogger.aAlarm[257].bRaised THEN
	EventLogger.aAlarm[257].Clear(0, TRUE);
END_IF


//Zusammenfassung Störungen
bStoerung := FALSE;
nStoerungsgrund := 0;
FOR i:=1 TO Parameter.cAnzEvents DO
	IF			EventLogger.aAlarm[i].bRaised THEN
		bStoerung := TRUE;
		nStoerungsgrund := i;
		EventLogger.aAlarm[i].RequestEventText(2055, sText, SIZEOF(sText));		
		//UTF8_TO_STRING(pDstSTRING := ADR(sFehlerText), pSrcUTF8 := ADR(sText), nDstsize := SIZEOF(sFehlerText));
		sFehlerText := sText;
	END_IF
END_FOR

IF		NOT bStoerung THEN
	sFehlerText := '';
END_IF

IF			aStationInfo.bStoerung THEN
	bStoerung := TRUE;
END_IF


// Störungen der Überstromschutzklemmen
fb601A2();				
fb601A5();
IF			fb601A2.bStoerung 
		OR	fb601A5.bStoerung THEN
	bStoerung := TRUE;
END_IF

IF			bPosNachHbNio THEN
	bStoerung := TRUE;
END_IF

IF			bStoerung
	OR		bE_SafetyProgStop THEN
	fbTurmleuchte.stoerung();
END_IF


//***********************************************************************************************
//Warnungen
bWarnung := FALSE;
IF			aStationInfo.bWarnung THEN
	bWarnung := TRUE;
	fbTurmleuchte.warnung();
END_IF


//Maschinenstatus	(noch schön machen!) (lesen fertig und abgebrochen und so wird trozdem überschrieben)
IF			bE_Handbetrieb THEN
	HMI.StatusbarSetzen('Handbetrieb aktiviert', StatusbarFarbe.orange);
	sMqttStatus := 'handbetrieb';
ELSIF		bStoerung THEN
	
	IF			sFehlerText <> '' THEN
		HMI.StatusbarSetzen(sFehlerText, StatusbarFarbe.rot);
	ELSE
		HMI.StatusbarSetzen('Störung (Infos im Event Logger)', StatusbarFarbe.rot);
	END_IF
	IF			bPosNachHbNio THEN
		HMI.StatusbarSetzen('Falsche Position beim Verlassen des Handbetriebs (siehe Eventlogger)', StatusbarFarbe.rot);
	END_IF
	IF			fb601A2.bStoerung THEN
		HMI.StatusbarSetzen('Störung der Sicherungsklemme 601A2 (siehe Eventlogger)', StatusbarFarbe.rot);
	END_IF
	IF			fb601A5.bStoerung THEN
		HMI.StatusbarSetzen('Störung der Sicherungsklemme 601A5 (siehe Eventlogger)', StatusbarFarbe.rot);
	END_IF
	
	sMqttStatus := 'steht';
ELSIF		bWarnung THEN
	HMI.StatusbarSetzen('Eine Warnung steht an (Infos im Event Logger)', StatusbarFarbe.orange);
	sMqttStatus := 'warnung';
ELSIF		bProduzieren THEN
	sStatus := 'Produziert im Zyklusbetrieb';
	
	FOR	i := 0 TO nPunkte DO
		sStatus := CONCAT(sStatus, ' .');
	END_FOR	

	HMI.StatusbarSetzen(sStatus, StatusbarFarbe.gruen);
	sMqttStatus := 'produziert';
ELSE	
	IF			bInitBeendet THEN
		HMI.StatusbarSetzen('Bereit', StatusbarFarbe.gruen);
		sMqttStatus := 'bereit';
	ELSIF		(eInitStatus = InitStatus.bereit) THEN
		HMI.StatusbarSetzen('Bitte Initialisierung Starten (Blaue Taste betätigen)' , StatusbarFarbe.blau);
		sMqttStatus := 'init';
	ELSE
		sStatus := 'Initialisiert';
		
		FOR	i := 0 TO nPunkte DO
			sStatus := CONCAT(sStatus, ' .');
		END_FOR
		
		HMI.StatusbarSetzen(sStatus, StatusbarFarbe.gruen);
		sMqttStatus := 'init';
	END_IF
END_IF

//Punkte
fbStatusPunkteZeit(PT := T#300MS, IN := TRUE);
			
IF			fbStatusPunkteZeit.Q THEN
	IF			nPunkte < 5 THEN
		nPunkte := nPunkte+1;
	ELSE
		nPunkte := 0;
	END_IF
	fbStatusPunkteZeit(IN := FALSE);
END_IF


// Fehlermldung Safety neustarten
IF		NOT bE_SafetyInRun THEN
	IF 	NOT	EventLogger.aAlarm[100].bRaised THEN
		EventLogger.aAlarm[100].Raise(0);
	END_IF	
END_IF

IF			bE_SafetyInRun THEN
	IF		EventLogger.aAlarm[100].bRaised THEN
		EventLogger.aAlarm[100].Clear(0, TRUE);
	END_IF
END_IF

bA_Lampe_Schritt := MAIN.fbSt1.bSchrittbetriebAktiv AND MAIN.HMI.bProgrammgeladen;

safetyReset();
fbTurmleuchte();		
fbTurmleuchte.reset(); //Alle meldungen zurücksetzten, damit jeder Programmteil neue senden kann

METHOD auftragAnfordern	:ST_AufnahmeInfo
VAR_INPUT
END_VAR
VAR
	stAufnahmeInfo:			ST_AufnahmeInfo;
END_VAR
IF			(stStueckzaehler.nGutteileAuftrag >= ArtikelParam.akt.nAuftragsMenge)
	AND		(ArtikelParam.akt.nAuftragsMenge <> 0) THEN
	bStopNachZyklus := TRUE;
END_IF


IF			bStopNachZyklus THEN
	stAufnahmeInfo.stArtParam.sArtikel := '';
ELSE
	stAufnahmeInfo.stArtParam := ArtikelParam.akt;
END_IF

auftragAnfordern := stAufnahmeInfo;
END_METHOD

ACTION init:
CASE eInitStatus OF
	
	//********************************************************************************************************************
	InitStatus.bereit:	
				
		IF 		 	bE_NotHalt
			AND NOT bProgStop THEN 
			eInitStatus := InitStatus.luftdruck;
		END_IF
		
	//********************************************************************************************************************
	InitStatus.luftdruck:
		
		bA_Hauptventil := TRUE;
		
		IF			bE_LuftdruckIO THEN			
			eInitStatus := InitStatus.stationen;
			aStationInfo.bInit := TRUE;
		END_IF
		
	//********************************************************************************************************************
	InitStatus.stationen:
		
		eInitStatus := InitStatus.fertig;
		
		aStationInfo.bZyklusFertig := TRUE;		//RST gibts nicht, darum auf Zyklus fertig setzen
	
		IF		NOT aStationInfo.bInitBeendet THEN
			eInitStatus := InitStatus.stationen;
		END_IF

		
		
	//********************************************************************************************************************
	InitStatus.fertig:

		bInitBeendet := TRUE;
		
END_CASE
END_ACTION

ACTION Lampen:
//NotHalt
fbBlinkZeit(IN := NOT fbBlinkZeit.Q, PT:= T#400MS);

IF 			bE_LampeNotHalt THEN
	IF 			fbBlinkZeit.Q THEN
		bA_Lampe_NotHalt := NOT bA_Lampe_NotHalt;
	END_IF
ELSE
	bA_Lampe_NotHalt := bE_LampeNHReset;
END_IF

//NotHalt Reset
bA_Lampe_NHReset	:= bE_LampeNHReset;

//Start/Stop
bA_Lampe_Start 		:= 		bProduzieren AND NOT bStopNachZyklus 	OR 	bLampenTest;
bA_Lampe_Stop 		:= NOT 	bProduzieren 							OR 	bLampenTest;
//bA_Lampe_ProgStop 	:= 		bE_SafetyProgStop						OR 	bLampenTest;
bA_Lampe_Stoerung	:= 		bLampeStoerung							OR	bLampenTest;

//Bedienboxen


bLampeStoerung := FALSE;
END_ACTION

METHOD reset
VAR_INPUT
END_VAR
bProduzieren := FALSE;
eInitStatus := InitStatus.bereit;
bInitBeendet := FALSE;
END_METHOD

ACTION safetyReset:
//Safety Group Errorack.
CASE SafetyAck OF
	
    //********************************************
	1:         
		IF         	bE_SafetyComErr
			OR		bE_SafetyOtherErr  THEN
			   SafetyAck := SafetyAck + 1;
			   bA_SafetyRun := FALSE;
			   fbErrTP(IN := FALSE,PT:=T#0.5S);
		END_IF
		
	//********************************************			
	2:         
		fbErrTP(IN := TRUE,PT:=T#0.1S);
		IF                     NOT     fbErrTP.Q THEN
				   SafetyAck := SafetyAck + 1;
		END_IF
		
	//********************************************
	3:         
		fbErrTP(IN := FALSE,PT:=T#0.5S);
	   	bA_SafetyRun := TRUE;
		SafetyAck := 1;
                                   
END_CASE

bA_SafetyReset := fbErrTP.Q;
END_ACTION

METHOD zaehlerAusschuss : BOOL
VAR_INPUT
END_VAR
stStueckzaehler.nAusschussAuftrag 	:= stStueckzaehler.nAusschussAuftrag + 1;
stStueckzaehler.nAusschussTag 		:= stStueckzaehler.nAusschussTag + 1;
stStueckzaehler.nAusschussGesamt 	:= stStueckzaehler.nAusschussGesamt + 1;

stStueckzaehler.nAuftragszaehler	:= stStueckzaehler.nAuftragszaehler + 1;
stStueckzaehler.nGesamt				:= stStueckzaehler.nGesamt + 1;
END_METHOD

METHOD zaehlerGut : BOOL
VAR_INPUT
END_VAR
stStueckzaehler.nGutteileAuftrag 	:= stStueckzaehler.nGutteileAuftrag + 1;
stStueckzaehler.nGutteileTag 		:= stStueckzaehler.nGutteileTag + 1;
stStueckzaehler.nGutteileGesamt 	:= stStueckzaehler.nGutteileGesamt + 1;

stStueckzaehler.nAuftragszaehler	:= stStueckzaehler.nAuftragszaehler + 1;
stStueckzaehler.nGesamt				:= stStueckzaehler.nGesamt + 1;
END_METHOD

END_PROGRAM

// ---- POUs/FB_Hmi.TcPOU
FUNCTION_BLOCK FB_Hmi
VAR
	
	// FB
	fbDatei:			FB_Datei;
	bDateiSchreiben: BOOL;
	
	
	//Infostatusbar
	sStatus:				STRING(255);
	eStatusbarFarbe:		StatusbarFarbe := 0;
	
	nColorInfoBalken:		DWORD;
	
	//Programmauswahl		
	sArtikelProgrammTemp:	STRING; //InputTextbox	
	stQrCode:						ST_QrCode;

	bAuftragGeladen:		BOOL;

	//Vorwahlablauf
	eAblaufStatus:			AblaufStatus := AblaufStatus.bereit;
	//fbMessage:				FB_Message;	

	bWartungAnstehend:		BOOL;
	
	ProgrammLeer:			ST_Programme;
	aProgrammNamen:			ARRAY[1..Parameter.cMaxProgramme] OF STRING;
	
	bBtnProgrammSpeichern:	BOOL;
	bBtnProgrammLoeschen:	BOOL;
	bBtnProgrammAnzeigen:	BOOL;
	bBtnKonfigLeeren:		BOOL;
	bBtnDateiSchreiben:		BOOL;
	bBtnDateiLesen:			BOOL;
	
	//aAktorBew:		ARRAY [1..Parameter.cAnzSchritte] OF ST_AktorKonfig;
	//aAktorBewTemp:	ARRAY [1..Parameter.cAnzSchritte] OF ST_AktorKonfig;

	nFreierPlatz: 	INT;
	nNamenCheck: 	INT;
	i:				INT;
	
	bPopUpUeberschreiben:	BOOL;
	bPopUpLoeschen:			BOOL;
	bPopUpAnzeigen:			BOOL;
	bBtnPopUpJa: 			BOOL;
	bBtnPopUpNein:			BOOL;
	sPopUpText:				STRING;
	
	nPopUpXOffset:			INT;
	bBtnProgrammLaden:		BOOL;
	nEnumWandeln: 			INT;
	bProgrammeSchreiben: 	BOOL;
	bProgrammGeladen:		BOOL;
	nLetztesProgramm:		INT;
	bInit: 					BOOL := TRUE;
	bProgeammLadenBtnInaktiv: BOOL;
	bBtnSchrittbetrieb:	BOOL;
	
END_VAR

VAR_INPUT
	sQrCode:				STRING;
	bBtnAnzeigeStation:		BOOL;
	bProgrammAngewaehlt:	BOOL;
	ProgrammTemp:			ST_Programme;
END_VAR

VAR_OUTPUT
	nAnzeigeStation:		INT := 1;
	sStationStatus:			STRING;
	nAngewaehltesProg:		INT;
END_VAR


VAR_INPUT PERSISTENT
	aProgramm:				ARRAY[1..Parameter.cMaxProgramme] OF ST_Programme;
END_VAR

IF			bBtnAnzeigeStation THEN
	bBtnAnzeigeStation := FALSE;
	nAnzeigeStation := nAnzeigeStation + 1;
	IF			nAnzeigeStation > Parameter.cAnzStationen THEN
			nAnzeigeStation := 1;
	END_IF
END_IF

IF		nAnzeigeStation = 1 THEN
	sStationStatus := MAIN.fbSt1.sStationsStatus;
ELSIF	nAnzeigeStation = 2 THEN
	;
END_IF



// Wartung anstehend
(*
bWartungAnstehend := 	MAIN.fbSt1.bWarnungNothalt
					OR	MAIN.fbSt1.bWarnungZweiHand;
*)

//Programm abspeichern
CASE eAblaufStatus OF
	
	//***********************************************************************************************
	AblaufStatus.bereit: 
		//MAIN.fbWritePersistentData.START := FALSE;
		IF			bBtnProgrammSpeichern THEN
			bBtnProgrammSpeichern := FALSE;
			FOR i := 1 TO Parameter.cAnzAktoren DO
				ProgrammTemp.aAktorKonfig[i].tFahrZeit := UINT_TO_TIME(ProgrammTemp.aAktorKonfig[i].nFahrZeit);
				ProgrammTemp.aAktorKonfig[i].tHalteZeit := UINT_TO_TIME(ProgrammTemp.aAktorKonfig[i].nHalteZeit);
			END_FOR
			eAblaufStatus := AblaufStatus.nameUeberpruefen;
		ELSIF			bBtnProgrammLoeschen THEN
			bBtnProgrammLoeschen := FALSE;
			bPopUpLoeschen := TRUE;
			eAblaufStatus := AblaufStatus.programmLoeschen;
		ELSIF 			bBtnProgrammAnzeigen THEN
			bBtnProgrammAnzeigen := FALSE;
			eAblaufStatus := AblaufStatus.programmAnzeigen;
		END_IF
		
	//***********************************************************************************************	
	// Programmname vergleichen Rückgabewert: 1= Name nicht vergeben / X = Name vergeben Platznummer
	AblaufStatus.nameUeberpruefen:	
		nNamenCheck := 0;
		nNamenCheck :=	programmNameCheck();
		
		IF			(nNamenCheck = 999) THEN
			eAblaufStatus := AblaufStatus.freierPlatzsuchen;
		ELSE			
			// PopUp einblenden
			eAblaufStatus := AblaufStatus.popUp;
			bPopUpUeberschreiben := TRUE;
		END_IF
		
	//***********************************************************************************************	
	// Freier Programmplatz finden und speichern
	AblaufStatus.freierPlatzsuchen:
		
		nFreierPlatz := 0;
		nFreierPlatz := programmFreierPlatzSuchen();
		
		IF 		nFreierPlatz <> 0 THEN
			programmTempLaden();
			aProgramm[nFreierPlatz] := ProgrammTemp;
			programmNamenSchreiben();
			eAblaufStatus := AblaufStatus.bereit;
			bProgrammGeladen := FALSE;
			MAIN.bWritePersistentMan := TRUE;
		END_IF
		
	//***********************************************************************************************	
	// Freier Programmplatz finden
	AblaufStatus.popUp:	
	
		IF			bBtnPopUpNein THEN
			bBtnPopUpNein := FALSE;
			eAblaufStatus := AblaufStatus.bereit;
			bPopUpUeberschreiben := FALSE;
		ELSIF		bBtnPopUpJa THEN
			bBtnPopUpJa := FALSE;
			programmTempLaden();
			aProgramm[nNamenCheck] := ProgrammTemp;
			programmNamenSchreiben();
			eAblaufStatus := AblaufStatus.bereit;
			MAIN.bWritePersistentMan := TRUE;
			bProgrammGeladen := FALSE;
			bPopUpUeberschreiben := FALSE;
		END_IF
		
	//***********************************************************************************************	
	// Programm anzeigen
	AblaufStatus.programmAnzeigen:	
		
			nNamenCheck := 0;
			nNamenCheck :=	programmNameCheck();
			ProgrammTemp := aProgramm[nNamenCheck];
			eAblaufStatus := AblaufStatus.bereit;
		
	//***********************************************************************************************	
	// Programm löschen
	AblaufStatus.programmLoeschen:		
	
		IF			bBtnPopUpNein THEN
			bBtnPopUpNein := FALSE;
			bPopUpLoeschen := FALSE;
			eAblaufStatus := AblaufStatus.bereit;	
		ELSIF		bBtnPopUpJa THEN	
			bBtnPopUpJa := FALSE;
			bPopUpLoeschen := FALSE;
			nNamenCheck := 0;
			nNamenCheck :=	programmNameCheck();
			aProgramm[nNamenCheck] := ProgrammLeer;
			ProgrammTemp := ProgrammLeer;
			bProgrammGeladen := FALSE;
			programmeAufraeumen ();
			programmNamenSchreiben();
			MAIN.bWritePersistentMan := TRUE;
			eAblaufStatus := AblaufStatus.bereit;
		END_IF
	
END_CASE

// PopUp einblenden
IF			bPopUpUeberschreiben
	OR		bPopUpLoeschen THEN
	bPopUpAnzeigen := TRUE;
	nPopUpXOffset	:=	-800;			
ELSE
	bPopUpAnzeigen := FALSE;
	nPopUpXOffset	:= 0;
END_IF

IF			bPopUpUeberschreiben THEN
	sPopUpText := 'Soll das bestehende Programm überscherieben werden?';
ELSIF		bPopUpLoeschen THEN
	sPopUpText := 'Soll das angewählte Programm gelöscht werden?';
END_IF

//Programm laden
IF			bBtnProgrammLaden 
	AND		programmGueltig(nAngewaehltesProg) = 1 THEN
	ProgrammTemp := ProgrammLeer;
	ProgrammTemp := aProgramm[nAngewaehltesProg];
	IF		NOT bProgrammGeladen THEN
		MAIN.fbSt1.extReset();
	END_IF
	bProgrammGeladen := TRUE;
	nLetztesProgramm := nAngewaehltesProg;	
END_IF
IF			nLetztesProgramm <> nAngewaehltesProg THEN
	bProgrammGeladen := FALSE;
END_IF

IF			bBtnProgrammLaden
	AND		bProgrammGeladen THEN
	bBtnProgrammLaden := FALSE;
END_IF



// Prgramm laden Button inaktiv setzen
IF			NOT	MAIN.bInitBeendet 
		OR	NOT	(nAngewaehltesProg > 0) THEN
	bProgeammLadenBtnInaktiv := TRUE;
	bProgrammGeladen := FALSE;
ELSE
	bProgeammLadenBtnInaktiv := FALSE;
	
END_IF

// Programm laden
IF			(bBtnProgrammLaden 
	AND NOT bProgrammGeladen)
	OR 		bInit 	 
	OR		bBtnProgrammSpeichern THEN
	programmTempLaden();
	programmNamenSchreiben();
//	bProgrammAngewaehlt := TRUE;
	bBtnProgrammLaden := FALSE;
END_IF

// Programmmaske leeren
IF			bBtnKonfigLeeren THEN
	bBtnKonfigLeeren := FALSE;
	bProgrammgeladen := FALSE;
	bProgrammAngewaehlt := FALSE;
	ProgrammTemp := ProgrammLeer;
END_IF

// Schrittbetrieb
IF			bBtnSchrittbetrieb THEN
	MAIN.fbSt1.bSchrittbetriebAktiv := TRUE;
ELSE
	MAIN.fbSt1.bSchrittbetriebAktiv := FALSE;
END_IF

// Datei schreiben
IF			bDateiSchreiben THEN
	bDateiSchreiben := NOT fbDatei.schreiben();
END_IF


bInit := FALSE;

METHOD programmeAufraeumen : BOOL
VAR_INPUT
END_VAR

VAR
	i: INT;
	nErsterLeererPlatz: INT;
END_VAR
// Leerer Platz suchen
FOR i:=nAngewaehltesProg TO Parameter.cMaxProgramme DO
	aProgramm[i] := aProgramm[i+1];
END_FOR
END_METHOD

METHOD programmExport : BOOL
VAR_INPUT
END_VAR
END_METHOD

METHOD programmFreierPlatzSuchen : INT
VAR_INPUT
END_VAR

VAR
	i: INT;
END_VAR
FOR i := 1 TO Parameter.cMaxProgramme DO
	IF			aProgramm[i].sName = '' THEN
		programmFreierPlatzSuchen := i;
		EXIT;
	END_IF
END_FOR
END_METHOD

METHOD programmGueltig : INT
VAR_INPUT
	programmPlatz: INT;
END_VAR
// Ausgabe: 
// 1 = Programm gültig
// 2 = Programm ungültig

IF			aProgramm[programmPlatz].sName = '' THEN
	programmGueltig := 2;
ELSE
	programmGueltig := 1;
END_IF
END_METHOD

METHOD programmImport : BOOL
VAR_INPUT
END_VAR
END_METHOD

METHOD programmNameCheck : INT
VAR_INPUT
END_VAR

VAR
	i: INT;
END_VAR
// Sucht den eingegeben Programmnamen im Array
// Wenn der Name nicht gefunden wird der Rückgabewert 999 zurückgegeben
// wenn der Name gefunden wird wird der entsprechende Index zurückgegeben

FOR i := 1 TO Parameter.cMaxProgramme DO
	IF			ProgrammTemp.sName = aProgramm[i].sName THEN
		programmNameCheck := i;
		EXIT;
	ELSE
		programmNameCheck := 999;
	END_IF
END_FOR
END_METHOD

METHOD programmNamenSchreiben : BOOL
VAR_INPUT
END_VAR
FOR i := 1 TO Parameter.cMaxProgramme DO
	// Programmnamen von ProgrammArray in Namen Array kopieren, braucht es für die Combo Box Array
	aProgrammNamen[i] := aProgramm[i].sName; 
END_FOR
END_METHOD

METHOD programmTempLaden : BOOL
VAR_INPUT
END_VAR
VAR
	i: INT;
	j: INT;
END_VAR
FOR i := 1 TO Parameter.cMaxProgramme DO
	//DropDown INT in Enum wandeln
	FOR j := 1 TO Parameter.cAnzSchritte DO
		IF			ProgrammTemp.aAktorBew[j].nNummer = 0 THEN
			ProgrammTemp.aAktorBew[j].eAblaufStatus := AblaufStatus.default;
		ELSIF			ProgrammTemp.aAktorBew[j].nNummer = 1 THEN
			ProgrammTemp.aAktorBew[j].eAblaufStatus := AblaufStatus.aktor01Vor;
		ELSIF		ProgrammTemp.aAktorBew[j].nNummer = 2 THEN
			ProgrammTemp.aAktorBew[j].eAblaufStatus := AblaufStatus.aktor01Zurueck;
		ELSIF		ProgrammTemp.aAktorBew[j].nNummer = 3 THEN
			ProgrammTemp.aAktorBew[j].eAblaufStatus := AblaufStatus.aktor02Vor;
		ELSIF		ProgrammTemp.aAktorBew[j].nNummer = 4 THEN
			ProgrammTemp.aAktorBew[j].eAblaufStatus := AblaufStatus.aktor02Zurueck;
		ELSIF		ProgrammTemp.aAktorBew[j].nNummer = 5 THEN
			ProgrammTemp.aAktorBew[j].eAblaufStatus := AblaufStatus.aktor03Vor;
		ELSIF		ProgrammTemp.aAktorBew[j].nNummer = 6 THEN
			ProgrammTemp.aAktorBew[j].eAblaufStatus := AblaufStatus.aktor03Zurueck;
		ELSIF		ProgrammTemp.aAktorBew[j].nNummer = 7 THEN
			ProgrammTemp.aAktorBew[j].eAblaufStatus := AblaufStatus.aktor04Vor;
		ELSIF		ProgrammTemp.aAktorBew[j].nNummer = 8 THEN
			ProgrammTemp.aAktorBew[j].eAblaufStatus := AblaufStatus.aktor04Zurueck;
		ELSIF		ProgrammTemp.aAktorBew[j].nNummer = 9 THEN
			ProgrammTemp.aAktorBew[j].eAblaufStatus := AblaufStatus.aktor05Vor;
		ELSIF		ProgrammTemp.aAktorBew[j].nNummer = 10 THEN
			ProgrammTemp.aAktorBew[j].eAblaufStatus := AblaufStatus.aktor05Zurueck;
		ELSIF		ProgrammTemp.aAktorBew[j].nNummer = 11 THEN
			ProgrammTemp.aAktorBew[j].eAblaufStatus := AblaufStatus.aktor06Vor;
		ELSIF		ProgrammTemp.aAktorBew[j].nNummer = 12 THEN
			ProgrammTemp.aAktorBew[j].eAblaufStatus := AblaufStatus.aktor06Zurueck;
		ELSIF		ProgrammTemp.aAktorBew[j].nNummer = 13 THEN
			ProgrammTemp.aAktorBew[j].eAblaufStatus := AblaufStatus.teilAnwesend;
		ELSIF		ProgrammTemp.aAktorBew[j].nNummer = 14 THEN
			ProgrammTemp.aAktorBew[j].eAblaufStatus := AblaufStatus.extGeraetBereit;
		ELSIF		ProgrammTemp.aAktorBew[j].nNummer = 15 THEN
			ProgrammTemp.aAktorBew[j].eAblaufStatus := AblaufStatus.extGeraetStart;
		ELSIF		ProgrammTemp.aAktorBew[j].nNummer = 16 THEN
			ProgrammTemp.aAktorBew[j].eAblaufStatus := AblaufStatus.warten;
		END_IF
	END_FOR
END_FOR
END_METHOD

METHOD programmTempLoeschen : BOOL
VAR_INPUT
END_VAR
	ProgrammTemp.nNr := 0;
	ProgrammTemp.sName := '';
FOR	i := 1 TO Parameter.cAnzAktoren DO
	ProgrammTemp.aAktorKonfig[i].nSensArbeitsPos := 0;
	ProgrammTemp.aAktorKonfig[i].nSensRuhePos := 0;
	ProgrammTemp.aAktorKonfig[i].nFahrZeit := 0;
	ProgrammTemp.aAktorKonfig[i].tFahrZeit := T#0MS;
	ProgrammTemp.aAktorKonfig[i].nHalteZeit := 0;
	ProgrammTemp.aAktorKonfig[i].tHalteZeit := T#0MS;

END_FOR
END_METHOD

PROPERTY Status : STRING(255)
GET
Status := sStatus;
END_GET
SET
sStatus := Status;
END_SET
END_PROPERTY

METHOD StatusbarInfoSenden
VAR_INPUT
	sText : STRING;
	eColor : StatusbarFarbe;
END_VAR
Status := sText ;

//Farbe
CASE eColor OF
	StatusbarFarbe.gruen:	nColorInfoBalken := 16#FF39A64E;
	StatusbarFarbe.orange:	nColorInfoBalken := 16#FFFFA600;
	StatusbarFarbe.rot:		nColorInfoBalken := 16#FFE3001B;
END_CASE
END_METHOD

METHOD StatusbarSetzen : BOOL
VAR_INPUT
	sText : STRING;
	eColor : StatusbarFarbe;
END_VAR


Status := sText ;

//Farbe
CASE eColor OF
	StatusbarFarbe.gruen:	nColorInfoBalken := 16#FF39A64E;
	StatusbarFarbe.orange:	nColorInfoBalken := 16#FFFFA600;
	StatusbarFarbe.rot:		nColorInfoBalken := 16#FFE3001B;
	StatusbarFarbe.blau:	nColorInfoBalken := 16#FF0080FF;
END_CASE
END_METHOD

PROPERTY StatusFarbe : StatusbarFarbe
GET
StatusFarbe := eStatusbarFarbe;
END_GET
SET
eStatusbarFarbe := StatusFarbe;
END_SET
END_PROPERTY

END_FUNCTION_BLOCK

// ---- POUs/FB_Datei.TcPOU
FUNCTION_BLOCK FB_Datei
VAR_INPUT
END_VAR
VAR_OUTPUT
END_VAR
VAR
	eDateiSchreiben:		AblaufStatus := AblaufStatus.bereit;	
                            	
	sNetId: 					T_AmsNetId := '';	(* TwinCAT system network address *)
	nZaehler:					INT;

END_VAR

(*
Autor: 		PFS
Version:	1.0
Beschreibung:
Diese Klasse legt die Messdaten in einem CSV-File ab.
*)

//fbSystemZeit(	NETID := Main.sSrcNetId,
//				START := NOT fbSystemZeit.START); 
//schreibAblauf();

METHOD schreiben : BOOL
VAR_INPUT
	
END_VAR
VAR
END_VAR
VAR_INST
	sFileName: 					T_MaxString;(* CSV destination file path and name *)
	hFile:						UINT := 0;(* File handle of the source file *)
	                        	
	fbFileOpen:					FB_FileOpen;(* Opens file *)
	fbFileClose:				FB_FileClose;(* Closes file *)
	fbFilePuts:					FB_FilePuts;(* Writes one record (line) *)
	fbFileWrite:				FB_FileWrite; 
	
	
	sTempString:				STRING(255);
	sLine:						STRING(255);
	
	i:							INT;
	nIndex:						INT;
END_VAR
CASE eDateiSchreiben OF
	
	//***********************************************************************************************
	AblaufStatus.bereit:
	
		//Dateiname zusammensetzen
		sFileName := CONCAT(Parameter.sPfad, MAIN.HMI.ProgrammTemp.sName);
		sFileName := CONCAT(sFileName, '.csv');
		
		hFile			:= 0;
		eDateiSchreiben 	:= AblaufStatus.oeffnen;
		
	//***********************************************************************************************
	AblaufStatus.oeffnen:
	
		fbFileOpen( bExecute := FALSE  );
		
		fbFileOpen( 	sNetId := sNetId,
						sPathName := sFileName,
						nMode := FOPEN_MODEWRITE,
						ePath := PATH_GENERIC,
						bExecute := TRUE);
						
		eDateiSchreiben := AblaufStatus.wartenOffen;
		
	//***********************************************************************************************
	AblaufStatus.wartenOffen:
	
		fbFileOpen( bExecute := FALSE, hFile => hFile );
		IF NOT fbFileOpen.bBusy THEN
			IF NOT fbFileOpen.bError THEN
				eDateiSchreiben := AblaufStatus.schreiben;
				sLine := '';
				nIndex := 0;
			ELSE	
				eDateiSchreiben := AblaufStatus.error;
			END_IF
		END_IF
				
	//***********************************************************************************************	
	AblaufStatus.schreiben:
	
//		FOR i := nIndex TO Parameter.cZyklenProMessung DO
			
//			sTempString := CONCAT(REAL_TO_STRING(aMessdaten[1,i].x), ';');
//			sTempString := CONCAT(sTempString, REAL_TO_STRING(aMessdaten[1,i].y));
//			sTempString := CONCAT(sTempString, '$R');
//			nIndex := i;
			
//			IF 			(LEN(sLine) + LEN(sTempString) <= 255) THEN
//				sLine := CONCAT(sLine, sTempString);
//			ELSE
//				EXIT;
//			END_IF
//		END_FOR
		
	
		fbFileWrite( bExecute := FALSE );
		
		fbFileWrite( sNetId := sNetId,
					hFile := hFile,
					pWriteBuff := ADR(MAIN.HMI.ProgrammTemp),
					cbWriteLen := SIZEOF(MAIN.HMI.ProgrammTemp),
					tTimeout := T#2S,    
					bExecute := TRUE );
		eDateiSchreiben := AblaufStatus.wartenGeschrieben;

	//***********************************************************************************************
	AblaufStatus.wartenGeschrieben:
	
		fbFileWrite( bExecute := FALSE);
		IF NOT fbFileWrite.bBusy THEN
			IF NOT fbFileWrite.bError THEN
				
				eDateiSchreiben := AblaufStatus.schliessen;(* Write next record *)
				
			ELSE(* Error *)
				eDateiSchreiben := AblaufStatus.error;
			END_IF
		END_IF

	//***********************************************************************************************
	AblaufStatus.schliessen:
	
		fbFileClose( bExecute := FALSE );
		fbFileClose( sNetId := sNetId, hFile := hFile, bExecute := TRUE );
		eDateiSchreiben := AblaufStatus.wartenGeschlossen;

	//***********************************************************************************************
	AblaufStatus.wartenGeschlossen:
	
		fbFileClose( bExecute := FALSE);
		IF ( NOT fbFileClose.bBusy ) THEN

			eDateiSchreiben := AblaufStatus.error;
		
			hFile := 0;
			
		END_IF

	//***********************************************************************************************
	AblaufStatus.error:
	
		IF ( hFile <> 0 ) THEN
			eDateiSchreiben := AblaufStatus.schliessen;
		ELSE
			eDateiSchreiben := AblaufStatus.bereit;
			schreiben := TRUE;
		END_IF
END_CASE
END_METHOD

END_FUNCTION_BLOCK

// ---- POUs/FB_Turmleuchte.TcPOU
FUNCTION_BLOCK FB_Turmleuchte
VAR_INPUT
END_VAR
VAR_OUTPUT
END_VAR
VAR
	bA_Summer					AT%Q*:BOOL;
	bA_LampeGruen				AT%Q*:BOOL;
	bA_LampeOrange				AT%Q*:BOOL;
	bA_LampeRot					AT%Q*:BOOL;
	bA_Zaehlen					AT%Q*:BOOL;
	
	tZaehlImpuls:				TP;
	
	bStoerung:					BOOL;
	bWarnung:					BOOL;
	bBetrieb:					BOOL;
	bZaehlen:					BOOL;
	
	bBtnSireneAktivieren:		BOOL;
END_VAR

VAR PERSISTENT
	bSireneAktiviert:			BOOL;
END_VAR

bA_LampeGruen := bBetrieb;
bA_LampeOrange :=bWarnung;
bA_LampeRot := bStoerung;
bA_Summer := bStoerung AND NOT MAIN.bProgStop AND MAIN.bProduzieren AND bSireneAktiviert;

IF			bZaehlen THEN
	tZaehlImpuls.IN := TRUE;
	bZaehlen := FALSE;
ELSE
	tZaehlImpuls.IN := FALSE;
END_IF


tZaehlImpuls(Q => bA_Zaehlen, PT := T#300MS);

IF			bBtnSireneAktivieren THEN
	bBtnSireneAktivieren := FALSE;
	bSireneAktiviert := NOT bSireneAktiviert;
END_IF

METHOD betrieb
VAR_INPUT
END_VAR
bBetrieb := true;
END_METHOD

METHOD reset : BOOL
VAR_INPUT
END_VAR
bStoerung := FALSE;
bWarnung := FALSE;
bBetrieb := FALSE;
END_METHOD

METHOD stoerung
VAR_INPUT
END_VAR
bStoerung := true;
END_METHOD

METHOD warnung
VAR_INPUT
END_VAR
bWarnung := true;
END_METHOD

METHOD zaehlen
VAR_INPUT
END_VAR
bZaehlen := true;
END_METHOD

END_FUNCTION_BLOCK

// ---- POUs/FB_Station01.TcPOU
FUNCTION_BLOCK FB_Station01 EXTENDS FB_Station IMPLEMENTS IF_Station
VAR_INPUT
	//Ablauf
	//aReihenfolge:	ARRAY [1..Parameter.cAnzSchritte] OF AblaufStatus;  // über HMI befüllen
	aReihenfolge:	ARRAY [1..Parameter.cAnzSchritte] OF ST_Reihenfolge;
	fbAktor:		ARRAY [1..Parameter.cAnzAktoren] OF FB_Aktor[
											(bSensAPVorhanden:= FALSE, 
											bSensRPVorhanden:= FALSE, 
											tZeitRP:= T#3000MS, 
											tZeitAP:= T#3000MS, 
											nErrorIdAP:= 13, 
											nErrorIdRP:= 14, 
											sBezeichnung:= 'Aktor 1'),
											
											(bSensAPVorhanden:= FALSE, 
											bSensRPVorhanden:= FALSE, 
											tZeitRP:= T#3000MS, 
											tZeitAP:= T#3000MS, 
											nErrorIdAP:= 15, 
											nErrorIdRP:= 16, 
											sBezeichnung:= 'Aktor 2'),
											
											(bSensAPVorhanden:= FALSE, 
											bSensRPVorhanden:= FALSE, 
											tZeitRP:= T#3000MS, 
											tZeitAP:= T#3000MS, 
											nErrorIdAP:= 17, 
											nErrorIdRP:= 18, 
											sBezeichnung:= 'Aktor 3'),
											
											(bSensAPVorhanden:= FALSE, 
											bSensRPVorhanden:= FALSE, 
											tZeitRP:= T#3000MS, 
											tZeitAP:= T#3000MS, 
											nErrorIdAP:= 19, 
											nErrorIdRP:= 20, 
											sBezeichnung:= 'Aktor 4'),
											
											(bSensAPVorhanden:= FALSE, 
											bSensRPVorhanden:= FALSE, 
											tZeitRP:= T#3000MS, 
											tZeitAP:= T#3000MS, 
											nErrorIdAP:= 21, 
											nErrorIdRP:= 22, 
											sBezeichnung:= 'Aktor 5'),
											
											(bSensAPVorhanden:= FALSE, 
											bSensRPVorhanden:= FALSE, 
											tZeitRP:= T#3000MS, 
											tZeitAP:= T#3000MS, 
											nErrorIdAP:= 23, 
											nErrorIdRP:= 24, 
											sBezeichnung:= 'Aktor 6')
											];
	bSchrittbetriebAktiv:	BOOL;
	sNaechsterSchritt:		STRING;
END_VAR
VAR_OUTPUT
END_VAR
VAR


	
	//Inputs	
	bE_extGeraetBereit			AT%I*:	BOOL;

	bE_Sensor					AT %I* : ARRAY[1..8] OF BOOL;
	bA_extGeraetStart			AT%Q*:	BOOL;
	//Outputs

	//FBs	

	
	// Not-Halt testen täglich
	bNotHaltTestIO:			BOOL;
	fbNotHaltGedrueckt:		R_TRIG;
	bBtnResetWarnNothalt:	BOOL;
	bWarnungNothalt:		BOOL;
	bBtnResetAuftrZaehler:	BOOL;
	fbFlankeSchritt:		R_TRIG;
	bInit:					BOOL := TRUE;
	iSchritt:				INT := 1;								
	i: 						INT;
	x: 						INT;
	bSensorTeilAnwesend: 	BOOL;
	nStatusSchritt: 		INT;
	nZyklusZaehler:			INT;	
	
END_VAR

VAR_OUTPUT
	sStationsStatus:	STRING;
END_VAR

VAR PERSISTENT
	nMonatVorher:			WORD;
	nTagVorher:				WORD;
	nZaehlerNotHalt:		DINT;
END_VAR

fbFlankeSchritt(CLK := MAIN.bE_Taste_Schritt AND bSchrittbetriebAktiv);

//Array "aReihenfolge" mit dem Ablauf befüllen
IF			MAIN.HMI.bProgrammAngewaehlt 
		AND	reihenfolgeSchreiben() THEN
	MAIN.HMI.bProgrammAngewaehlt := FALSE;
END_IF

//********************************************************************************	
//Aktoren
fbAktor[1](fbSchrittbetrieb := fbSchrittbetrieb);
fbAktor[2](fbSchrittbetrieb := fbSchrittbetrieb);
fbAktor[3](fbSchrittbetrieb := fbSchrittbetrieb);
fbAktor[4](fbSchrittbetrieb := fbSchrittbetrieb);
fbAktor[5](fbSchrittbetrieb := fbSchrittbetrieb);
fbAktor[6](fbSchrittbetrieb := fbSchrittbetrieb); 



FOR x := 1 TO Parameter.cAnzAktoren DO
	IF			MAIN.HMI.ProgrammTemp.aAktorKonfig[x].nSensRuhePos > 0 THEN			
		fbAktor[x].bE_sensRP 	:= bE_Sensor[MAIN.HMI.ProgrammTemp.aAktorKonfig[x].nSensRuhePos];
		fbAktor[x].bSensRPVorhanden := TRUE;
	ELSE
		fbAktor[x].bSensRPVorhanden := FALSE;
	END_IF
	IF			MAIN.HMI.ProgrammTemp.aAktorKonfig[x].nSensArbeitsPos > 0 THEN			
		fbAktor[x].bE_sensAP 	:= bE_Sensor[MAIN.HMI.ProgrammTemp.aAktorKonfig[x].nSensArbeitsPos];
		fbAktor[x].bSensAPVorhanden := TRUE;
	ELSE
		fbAktor[x].bSensAPVorhanden := FALSE;
	END_IF	
	IF			MAIN.HMI.ProgrammTemp.aAktorKonfig[x].tFahrZeit = T#0MS THEN
		fbAktor[x].tZeitRP 		:= T#2000MS;
		fbAktor[x].tZeitAP 		:= T#2000MS;
	ELSE
		fbAktor[x].tZeitRP 		:= MAIN.HMI.ProgrammTemp.aAktorKonfig[x].tFahrZeit;
		fbAktor[x].tZeitAP 		:= MAIN.HMI.ProgrammTemp.aAktorKonfig[x].tFahrZeit;
	END_IF
	
	
END_FOR
	IF			bE_Sensor[MAIN.HMI.ProgrammTemp.nTeilAnw] THEN
		bSensorTeilAnwesend := TRUE;
	ELSE
		bSensorTeilAnwesend := FALSE;
	END_IF

FOR x := 1 TO Parameter.cAnzAktoren DO
	IF			NOT	stStationInfo.bInitBeendet THEN
		fbAktor[x].bSensRPVorhanden := FALSE;
		fbAktor[x].bSensAPVorhanden := FALSE;
	END_IF
END_FOR
		
//********************************************************************************	
//Sonstige FBs


//********************************************************************************
//Basisklasse ausführen
SUPER^(	stStationInfo := stStationInfo);


//********************************************************************************
//Stoerungen
stStationInfo.bStoerung := 			(fbAktor[1].bStoerung
							OR		fbAktor[2].bStoerung
							OR		fbAktor[3].bStoerung
							OR		fbAktor[4].bStoerung
							OR		fbAktor[5].bStoerung
							OR		fbAktor[6].bStoerung)
							AND		Main.bProduzieren
							AND NOT Main.bE_Handbetrieb;
							
sStationsStatus := stStationInfo.sStatus;

//********************************************************************************
//Warnung
stStationInfo.bWarnung := (			FALSE);

//Not-Halt-Test nach einem Tag zurücksetzen
IF		 	(nTagVorher <> MAIN.fbSystemZeit.TIMESTR.wDay 
	OR 	  	nMonatVorher <> MAIN.fbSystemZeit.TIMESTR.wMonth)
	AND		MAIN.fbSystemZeit.TIMESTR.wMonth > 0 THEN		//Damit der fbSystemzeit sicher ausgeführt wurde
	nTagVorher := MAIN.fbSystemZeit.TIMESTR.wDay;
	nMonatVorher := MAIN.fbSystemZeit.TIMESTR.wMonth;
	bNotHaltTestIO := FALSE;

END_IF

	// Not-Halt wurde betätigt
	IF		NOT	bNotHaltTestIO 
		AND	NOT	MAIN.bE_NotHalt THEN
		bNotHaltTestIO := TRUE;
	END_IF
	
	//Fehlermeldung
	IF		NOT bNotHaltTestIO
		AND	NOT	EventLogger.aAlarm[40].bRaised THEN
		EventLogger.aAlarm[40].Raise(0);
	ELSIF		bNotHaltTestIO
		AND		EventLogger.aAlarm[40].bRaised THEN
		EventLogger.aAlarm[40].Clear(0, TRUE);
	END_IF
	// Not-Halt Wartung
	fbNotHaltGedrueckt(CLK := NOT(MAIN.bE_NotHalt) AND MAIN.bInitBeendet);
	IF		fbNotHaltGedrueckt.Q THEN
		nZaehlerNotHalt := nZaehlerNotHalt + 1;
	END_IF
	IF		nZaehlerNotHalt >= Parameter.cMaxZyklNotHalt 
			AND	NOT	bWarnungNothalt THEN
		bWarnungNothalt := TRUE;
	END_IF
	
	IF		bBtnResetWarnNothalt 
		AND bWarnungNothalt THEN
			bBtnResetWarnNothalt := FALSE;
			bWarnungNothalt := FALSE;
			nZaehlerNotHalt := 0;
	END_IF

// Auftragszähler Reset
IF			bBtnResetAuftrZaehler THEN
	bBtnResetAuftrZaehler := FALSE;
	MAIN.stStueckzaehler.nAusschussAuftrag 	:= 0;
	MAIN.stStueckzaehler.nGutteileAuftrag 	:= 0;
END_IF

// Nächster Schritt auf HMI anzeigen im Schrittbetrieb

CASE aReihenfolge[iSchritt].eAblauf OF
	AblaufStatus.default:			sNaechsterSchritt := 'default';
	AblaufStatus.aktor01Vor:		sNaechsterSchritt := 'Aktor 1 vor';
	AblaufStatus.aktor01Zurueck:	sNaechsterSchritt := 'Aktor 1 zurück';
	AblaufStatus.aktor02Vor:		sNaechsterSchritt := 'Aktor 2 vor';
	AblaufStatus.aktor02Zurueck:	sNaechsterSchritt := 'Aktor 2 zurück';
	AblaufStatus.aktor03Vor:		sNaechsterSchritt := 'Aktor 3 vor';
	AblaufStatus.aktor03Zurueck:	sNaechsterSchritt := 'Aktor 3 zurück';
	AblaufStatus.aktor04Vor:		sNaechsterSchritt := 'Aktor 4 vor';
	AblaufStatus.aktor04Zurueck:	sNaechsterSchritt := 'Aktor 4 zurück';
	AblaufStatus.aktor05Vor:		sNaechsterSchritt := 'Aktor 5 vor';
	AblaufStatus.aktor05Zurueck:	sNaechsterSchritt := 'Aktor 5 zurück';
	AblaufStatus.aktor06Vor:		sNaechsterSchritt := 'Aktor 6 vor';
	AblaufStatus.aktor06Zurueck:	sNaechsterSchritt := 'Aktor 6 zurück';
	AblaufStatus.teilAnwesend:		sNaechsterSchritt := 'teilAnwesend';
	AblaufStatus.bereit:			sNaechsterSchritt := 'bereit';
	AblaufStatus.error:				sNaechsterSchritt := 'error';
	AblaufStatus.extGeraetBereit:	sNaechsterSchritt := 'extGeraetBereit';
	AblaufStatus.extGeraetFertig:	sNaechsterSchritt := 'extGeraetFertig';
	AblaufStatus.extGeraetStart:	sNaechsterSchritt := 'extGeraetStart';
	AblaufStatus.fertig:			sNaechsterSchritt := 'fertig';
	AblaufStatus.warten:			sNaechsterSchritt := 'warten';
END_CASE



//************************************************************************
//Muss alles nach dem Ablauf sein, damit das Main die Aktuellen Werte hat.
//************************************************************************

//Zyklus Fertig	
stStationInfo.bZyklusFertig :=		NOT bTeilBearbeiten;
bInit := FALSE;

METHOD ablaufSchreiben : AblaufStatus
VAR_INPUT
END_VAR

VAR
	eAblaufStatus: AblaufStatus;
	i:		INT := 1;
END_VAR

// Ablauf aus ARRAY Reihenfolge in AblaufStatus schreiben
// Wenn beim Aktor Pendelbetrieb aktiviert ist, muss der Ablaufstatus jedes Mal wechseln zwischen den Zyklen, z.B. aktor01Vor <> aktor02Zurueck
// Dies wird z.B bei einer Verdrillvorrichtung für den RST benötigt
// MAIN.HMI.ProgrammTemp.aAktorKonfig[1]


IF			nZyklusZaehler = 0 THEN
	// Ablauf für Aktoren korrigieren gemäss ihrem aktuellen Zustand
		IF			fbAktor[1].inAP()
			AND		aReihenfolge[iSchritt].eAblauf = AblaufStatus.aktor01Vor THEN
				eAblaufStatus := AblaufStatus.aktor01Zurueck;
//		ELSIF 		fbAktor[1].inRP()
//			AND		aReihenfolge[iSchritt].eAblauf = AblaufStatus.aktor01Zurueck THEN
//				eAblaufStatus := AblaufStatus.aktor01Vor;
				
		ELSIF 		fbAktor[2].inAP()
			AND		aReihenfolge[iSchritt].eAblauf = AblaufStatus.aktor02Vor THEN
				eAblaufStatus := AblaufStatus.aktor02Zurueck;
//		ELSIF 		fbAktor[2].inRP()
//			AND		aReihenfolge[iSchritt].eAblauf = AblaufStatus.aktor02Zurueck THEN
//				eAblaufStatus := AblaufStatus.aktor02Vor;
		
		ELSIF 		fbAktor[3].inAP()
			AND		aReihenfolge[iSchritt].eAblauf = AblaufStatus.aktor03Vor THEN
				eAblaufStatus := AblaufStatus.aktor03Zurueck;
				
		ELSIF 		fbAktor[4].inAP()
			AND		aReihenfolge[iSchritt].eAblauf = AblaufStatus.aktor04Vor THEN
				eAblaufStatus := AblaufStatus.aktor04Zurueck;
				
		ELSIF 		fbAktor[5].inAP()
			AND		aReihenfolge[iSchritt].eAblauf = AblaufStatus.aktor05Vor THEN
				eAblaufStatus := AblaufStatus.aktor05Zurueck;
				
		ELSIF 		fbAktor[6].inAP()
			AND		aReihenfolge[iSchritt].eAblauf = AblaufStatus.aktor06Vor THEN
				eAblaufStatus := AblaufStatus.aktor06Zurueck;
				
		ELSE
			eAblaufStatus := aReihenfolge[iSchritt].eAblauf;
		END_IF


	//eAblaufStatus := aReihenfolge[iSchritt].eAblauf;
	aReihenfolge[iSchritt].eLetzterStatus := eAblaufStatus;
	
ELSE
	CASE aReihenfolge[iSchritt].eLetzterStatus OF
		
		//****************************************************************************************	
		//****************************************************************************************
		AblaufStatus.aktor01Vor:
			IF			MAIN.HMI.ProgrammTemp.aAktorKonfig[1].bReversierBetrieb THEN
				eAblaufStatus := AblaufStatus.aktor01Zurueck;
			ELSE
				eAblaufStatus := AblaufStatus.aktor01Vor;
			END_IF
			aReihenfolge[iSchritt].eLetzterStatus := eAblaufStatus;
			
		//****************************************************************************************	
		AblaufStatus.aktor01Zurueck:
			IF			MAIN.HMI.ProgrammTemp.aAktorKonfig[1].bReversierBetrieb THEN
				eAblaufStatus := AblaufStatus.aktor01Vor;
			ELSE
				eAblaufStatus := AblaufStatus.aktor01Zurueck;
			END_IF
			aReihenfolge[iSchritt].eLetzterStatus := eAblaufStatus;
			
		//****************************************************************************************	
		//****************************************************************************************
		AblaufStatus.aktor02Vor:
			IF			MAIN.HMI.ProgrammTemp.aAktorKonfig[2].bReversierBetrieb THEN
				eAblaufStatus := AblaufStatus.aktor02Zurueck;
			ELSE
				eAblaufStatus := AblaufStatus.aktor02Vor;
			END_IF
			aReihenfolge[iSchritt].eLetzterStatus := eAblaufStatus;
			
		//****************************************************************************************	
		AblaufStatus.aktor02Zurueck:
			IF			MAIN.HMI.ProgrammTemp.aAktorKonfig[2].bReversierBetrieb THEN
				eAblaufStatus := AblaufStatus.aktor02Vor;
			ELSE
				eAblaufStatus := AblaufStatus.aktor02Zurueck;
			END_IF	
			aReihenfolge[iSchritt].eLetzterStatus := eAblaufStatus;
			
		//****************************************************************************************	
		//****************************************************************************************
		AblaufStatus.aktor03Vor:
			IF			MAIN.HMI.ProgrammTemp.aAktorKonfig[3].bReversierBetrieb THEN
				eAblaufStatus := AblaufStatus.aktor03Zurueck;
			ELSE
				eAblaufStatus := AblaufStatus.aktor03Vor;
			END_IF
			aReihenfolge[iSchritt].eLetzterStatus := eAblaufStatus;
			
		//****************************************************************************************	
		AblaufStatus.aktor03Zurueck:
			IF			MAIN.HMI.ProgrammTemp.aAktorKonfig[3].bReversierBetrieb THEN
				eAblaufStatus := AblaufStatus.aktor03Vor;
			ELSE
				eAblaufStatus := AblaufStatus.aktor03Zurueck;
			END_IF
			aReihenfolge[iSchritt].eLetzterStatus := eAblaufStatus;
			
		//****************************************************************************************	
		//****************************************************************************************
		AblaufStatus.aktor04Vor:
			IF			MAIN.HMI.ProgrammTemp.aAktorKonfig[4].bReversierBetrieb THEN
				eAblaufStatus := AblaufStatus.aktor04Zurueck;
			ELSE
				eAblaufStatus := AblaufStatus.aktor04Vor;
			END_IF
			aReihenfolge[iSchritt].eLetzterStatus := eAblaufStatus;
			
		//****************************************************************************************	
		AblaufStatus.aktor04Zurueck:
			IF			MAIN.HMI.ProgrammTemp.aAktorKonfig[4].bReversierBetrieb THEN
				eAblaufStatus := AblaufStatus.aktor04Vor;
			ELSE
				eAblaufStatus := AblaufStatus.aktor04Zurueck;
			END_IF
			aReihenfolge[iSchritt].eLetzterStatus := eAblaufStatus;
			
		//****************************************************************************************	
		//****************************************************************************************
		AblaufStatus.aktor05Vor:
			IF			MAIN.HMI.ProgrammTemp.aAktorKonfig[5].bReversierBetrieb THEN
				eAblaufStatus := AblaufStatus.aktor05Zurueck;
			ELSE
				eAblaufStatus := AblaufStatus.aktor05Vor;
			END_IF
			aReihenfolge[iSchritt].eLetzterStatus := eAblaufStatus;
			
		//****************************************************************************************	
		AblaufStatus.aktor05Zurueck:
			IF			MAIN.HMI.ProgrammTemp.aAktorKonfig[5].bReversierBetrieb THEN
				eAblaufStatus := AblaufStatus.aktor05Vor;
			ELSE
				eAblaufStatus := AblaufStatus.aktor05Zurueck;
			END_IF
			aReihenfolge[iSchritt].eLetzterStatus := eAblaufStatus;
			
		//****************************************************************************************	
		//****************************************************************************************
		AblaufStatus.aktor06Vor:
			IF			MAIN.HMI.ProgrammTemp.aAktorKonfig[6].bReversierBetrieb THEN
				eAblaufStatus := AblaufStatus.aktor06Zurueck;
			ELSE
				eAblaufStatus := AblaufStatus.aktor06Vor;
			END_IF
			aReihenfolge[iSchritt].eLetzterStatus := eAblaufStatus;
			
		//****************************************************************************************	
		AblaufStatus.aktor06Zurueck:
			IF			MAIN.HMI.ProgrammTemp.aAktorKonfig[6].bReversierBetrieb THEN
				eAblaufStatus := AblaufStatus.aktor06Vor;
			ELSE
				eAblaufStatus := AblaufStatus.aktor06Zurueck;
			END_IF
			aReihenfolge[iSchritt].eLetzterStatus := eAblaufStatus;	
	ELSE
			eAblaufStatus := aReihenfolge[iSchritt].eAblauf;
			
	END_CASE	
END_IF


ablaufSchreiben := eAblaufStatus;
END_METHOD

METHOD init : BOOL
CASE eInitStatus OF
	//***********************************************************************************************
	InitStatus.bereit:
			
		IF 		NOT stStationInfo.bInitBeendet THEN
			EventLogger.aMessage[10].ipArguments.Clear().AddString('Aktoren');
			EventLogger.aMessage[10].Send(0);
			bTeilBearbeiten := FALSE;									// Hier richtig?
			eInitStatus := InitStatus.aktor1;
		END_IF
		
	//***********************************************************************************************
	InitStatus.aktor1:
		
		IF		fbAktor[1].ruhePos() THEN
			eInitStatus := InitStatus.aktor2;
		END_IF

	//***********************************************************************************************
	InitStatus.aktor2:
	
		IF		fbAktor[2].ruhePos() THEN
			eInitStatus := InitStatus.aktor3;
		END_IF

	//***********************************************************************************************
	InitStatus.aktor3:
	
		IF		fbAktor[3].ruhePos() THEN
			eInitStatus := InitStatus.aktor4;
		END_IF

	//***********************************************************************************************
	InitStatus.aktor4:
	
		IF		fbAktor[4].ruhePos() THEN
			eInitStatus := InitStatus.aktor5;
		END_IF

	//***********************************************************************************************
	InitStatus.aktor5:
	
		IF		fbAktor[5].ruhePos() THEN
			eInitStatus := InitStatus.aktor6;
		END_IF

	//***********************************************************************************************
	InitStatus.aktor6:	
	
		IF		fbAktor[6].ruhePos() THEN
			eInitStatus := InitStatus.fertig;
		END_IF
	
	//***********************************************************************************************
	InitStatus.fertig:
		
		EventLogger.aMessage[11].Send(0);
		
		stStationInfo.bInitBeendet := TRUE;
		MAIN.bProduzieren := FALSE;
		eInitStatus := InitStatus.bereit;
	
END_CASE

init := stStationInfo.bInitBeendet;
END_METHOD

METHOD reihenfolgeSchreiben : bool
VAR_INPUT
END_VAR
nZyklusZaehler := 0;

FOR i := 1 TO Parameter.cAnzSchritte DO	 	
	
	aReihenfolge[i].eAblauf := MAIN.HMI.ProgrammTemp.aAktorBew[i].eAblaufStatus;

	// Den Aktoren die Zeiten zuweisen aus dem Programm
	IF			aReihenfolge[i].eAblauf = Ablaufstatus.aktor01Vor
		OR		aReihenfolge[i].eAblauf = Ablaufstatus.aktor01Zurueck THEN
			aReihenfolge[i].tFahrzeit := MAIN.HMI.ProgrammTemp.aAktorKonfig[1].tFahrZeit;
			aReihenfolge[i].tHalteZeit := MAIN.HMI.ProgrammTemp.aAktorKonfig[1].tHalteZeit;
			
	ELSIF		aReihenfolge[i].eAblauf = Ablaufstatus.aktor02Vor
		OR		aReihenfolge[i].eAblauf = Ablaufstatus.aktor02Zurueck THEN
			aReihenfolge[i].tFahrzeit := MAIN.HMI.ProgrammTemp.aAktorKonfig[2].tFahrZeit;
			aReihenfolge[i].tHalteZeit := MAIN.HMI.ProgrammTemp.aAktorKonfig[2].tHalteZeit;
	
	ELSIF		aReihenfolge[i].eAblauf = Ablaufstatus.aktor03Vor
		OR		aReihenfolge[i].eAblauf = Ablaufstatus.aktor03Zurueck THEN
			aReihenfolge[i].tFahrzeit := MAIN.HMI.ProgrammTemp.aAktorKonfig[3].tFahrZeit;
			aReihenfolge[i].tHalteZeit := MAIN.HMI.ProgrammTemp.aAktorKonfig[3].tHalteZeit;
			
	ELSIF		aReihenfolge[i].eAblauf = Ablaufstatus.aktor04Vor
		OR		aReihenfolge[i].eAblauf = Ablaufstatus.aktor04Zurueck THEN
			aReihenfolge[i].tFahrzeit := MAIN.HMI.ProgrammTemp.aAktorKonfig[4].tFahrZeit;
			aReihenfolge[i].tHalteZeit := MAIN.HMI.ProgrammTemp.aAktorKonfig[4].tHalteZeit;
			
	ELSIF		aReihenfolge[i].eAblauf = Ablaufstatus.aktor05Vor
		OR		aReihenfolge[i].eAblauf = Ablaufstatus.aktor05Zurueck THEN
			aReihenfolge[i].tFahrzeit := MAIN.HMI.ProgrammTemp.aAktorKonfig[5].tFahrZeit;
			aReihenfolge[i].tHalteZeit := MAIN.HMI.ProgrammTemp.aAktorKonfig[5].tHalteZeit;
			
	ELSIF		aReihenfolge[i].eAblauf = Ablaufstatus.aktor06Vor
		OR		aReihenfolge[i].eAblauf = Ablaufstatus.aktor06Zurueck THEN
			aReihenfolge[i].tFahrzeit := MAIN.HMI.ProgrammTemp.aAktorKonfig[6].tFahrZeit;
			aReihenfolge[i].tHalteZeit := MAIN.HMI.ProgrammTemp.aAktorKonfig[6].tHalteZeit;
	END_IF
END_FOR	

reihenfolgeSchreiben := TRUE;
END_METHOD

METHOD reset : BOOL
CASE eResetStatus OF
	
	//***********************************************************************************************
	ResetStatus.bereit:
		
		eResetStatus := ResetStatus.ablaufAbbrechen;
		iSchritt := 1;
		
	//***********************************************************************************************
	ResetStatus.ablaufAbbrechen:
		
		eAblaufStatus 		:= AblaufStatus.bereit;
		fbSchrittbetrieb.reset();
		eResetStatus 		:= ResetStatus.aktoren;
	

		
	//***********************************************************************************************
	ResetStatus.aktoren:	
		FOR i:= 1 TO Parameter.cAnzAktoren DO
			fbAktor[i].bHandOverride := NOT MAIN.bE_SafetyProgStop;
			IF			fbAktor[i].ruhePos() THEN
				eResetStatus 		:= ResetStatus.fertig;
				fbAktor[i].bHandOverride := FALSE;
			END_IF
		END_FOR
	
	//***********************************************************************************************
	ResetStatus.fertig:
		
		eInitStatus := InitStatus.bereit;
		
		IF 			stStationInfo.bInitBeendet THEN		//Wenn schon initialisiert wurde, wird ein reinit durchgeführt
			stStationInfo.bInit := TRUE;				//War die Station schon am init, wurde bInit nie false und das init startet erneut
			stStationInfo.bInitBeendet := FALSE;
		END_IF
		
		reset := TRUE;
END_CASE
END_METHOD

METHOD teilBearbeiten : BOOL
VAR_INST
	//fbMessage:	FB_Message;
	fbTon:		TON;
	fbTonHalten:	TON;
	tTime:		TIME;
END_VAR
CASE eAblaufStatus OF
	
	AblaufStatus.bereit:
		IF			fbFlankeSchritt.Q 
			OR NOT	bSchrittbetriebAktiv THEN
			eAblaufStatus := AblaufStatus.schritt;
		END_IF
		
//****************************************************************************************
	AblaufStatus.schritt:		
		IF			aReihenfolge[iSchritt].eAblauf <> 	AblaufStatus.default  THEN
			eAblaufStatus := ablaufSchreiben();
			//eAblaufStatus := aReihenfolge[iSchritt].eAblauf;						// wird über Methode "ablaufSchreiben" erledigt
			fbTon(IN := FALSE, PT := aReihenfolge[iSchritt].tFahrzeit);		
			fbTonHalten(IN := FALSE, PT := aReihenfolge[iSchritt].tHaltezeit);	
		ELSE
			eAblaufStatus := AblaufStatus.fertig;
			nZyklusZaehler := nZyklusZaehler + 1;
			iSchritt := 1;
		END_IF
		
	//****************************************************************************************
	AblaufStatus.aktor01Vor:
	
		IF			fbAktor[1].arbeitsPos() THEN
			eAblaufStatus := AblaufStatus.naechsterSchritt;
		END_IF
	
	//****************************************************************************************
	AblaufStatus.aktor01Zurueck:
	
		IF			fbAktor[1].ruhePos() THEN
			eAblaufStatus := AblaufStatus.naechsterSchritt;
		END_IF
	
	//****************************************************************************************
	AblaufStatus.aktor02Vor:
	
		IF			fbAktor[2].arbeitsPos() THEN
			eAblaufStatus := AblaufStatus.naechsterSchritt;
		END_IF
	
	//****************************************************************************************
	AblaufStatus.aktor02Zurueck:
	
		IF			fbAktor[2].ruhePos() THEN
			eAblaufStatus := AblaufStatus.naechsterSchritt;
		END_IF

	//****************************************************************************************
	AblaufStatus.aktor03Vor:
	
		IF			fbAktor[3].arbeitsPos() THEN
			eAblaufStatus := AblaufStatus.naechsterSchritt;
		END_IF
	
	//****************************************************************************************
	AblaufStatus.aktor03Zurueck:
	
		IF			fbAktor[3].ruhePos() THEN
			eAblaufStatus := AblaufStatus.naechsterSchritt;
		END_IF

	//****************************************************************************************
	AblaufStatus.aktor04Vor:
	
		IF			fbAktor[4].arbeitsPos() THEN
			eAblaufStatus := AblaufStatus.naechsterSchritt;
		END_IF
	
	//****************************************************************************************
	AblaufStatus.aktor04Zurueck:
	
		IF			fbAktor[4].ruhePos() THEN
			eAblaufStatus := AblaufStatus.naechsterSchritt;
		END_IF

	//****************************************************************************************
	AblaufStatus.aktor05Vor:
	
		IF			fbAktor[5].arbeitsPos() THEN
			eAblaufStatus := AblaufStatus.naechsterSchritt;
		END_IF
	
	//****************************************************************************************
	AblaufStatus.aktor05Zurueck:	
	
		IF			fbAktor[5].ruhePos() THEN
			eAblaufStatus := AblaufStatus.naechsterSchritt;
		END_IF

	//****************************************************************************************
	AblaufStatus.aktor06Vor:
	
		IF			fbAktor[6].arbeitsPos() THEN
			eAblaufStatus := AblaufStatus.naechsterSchritt;
		END_IF
	
	//****************************************************************************************
	AblaufStatus.aktor06Zurueck:	
	
		IF			fbAktor[6].ruhePos() THEN
			eAblaufStatus := AblaufStatus.naechsterSchritt;
		END_IF
		
	//***********************************************************************************************
	AblaufStatus.warten:	
		
		fbTon(IN := TRUE);
		IF			fbton.Q THEN
			eAblaufStatus := AblaufStatus.naechsterSchritt;
		END_IF
		
	//***********************************************************************************************
	AblaufStatus.error:

			eAblaufStatus := AblaufStatus.naechsterSchritt;

	//***********************************************************************************************
	AblaufStatus.extGeraetBereit:

		IF		bE_extGeraetBereit	THEN
			eAblaufStatus := AblaufStatus.naechsterSchritt;
		END_IF
		
	//***********************************************************************************************
	AblaufStatus.extGeraetStart:
		
		bA_extGeraetStart := TRUE;
		IF		NOT	bE_extGeraetBereit	THEN
			eAblaufStatus := AblaufStatus.extGeraetFertig;		
		END_IF	
		
	//***********************************************************************************************
	AblaufStatus.extGeraetFertig:
		IF		bE_extGeraetBereit	THEN
			eAblaufStatus := AblaufStatus.naechsterSchritt;
			bA_extGeraetStart := FALSE;
		END_IF
			
	//***********************************************************************************************		
	AblaufStatus.teilAnwesend:
		
		IF			bSensorTeilAnwesend THEN
			eAblaufStatus := AblaufStatus.naechsterSchritt;	
		END_IF
	
	//***********************************************************************************************
	AblaufStatus.naechsterSchritt:
	
		fbTonHalten(IN := TRUE);
		IF			fbTonHalten.Q 
			AND NOT	MAIN.bE_Taste_Schritt THEN
			iSchritt := iSchritt + 1;
			eAblaufStatus := AblaufStatus.bereit;
		END_IF
		
	//***********************************************************************************************
	AblaufStatus.fertig:		
	
			eAblaufStatus := AblaufStatus.bereit;
			teilbearbeiten := TRUE;
			MAIN.bProduzieren := FALSE;
			MAIN.zaehlerGut();
		
END_CASE
END_METHOD

END_FUNCTION_BLOCK

// ---- POUs/StdStationen/FB_Station.TcPOU
FUNCTION_BLOCK FB_Station
VAR_INPUT
	ifStation:				IF_Station;
	bRstInPos: 				BOOL;
END_VAR
VAR_IN_OUT
	stStationInfo:			ST_Station;
END_VAR
VAR	
	//FBs	
	fbSchrittbetrieb:		FB_Schrittbetrieb;
								
	//Reset
	eResetStatus:			ResetStatus := ResetStatus.bereit;
	bBtnReset:				BOOL;
		
	//Sonstiges
	eInitStatus:			InitStatus := InitStatus.bereit;
	eAblaufStatus:			AblaufStatus := AblaufStatus.bereit;
	
	bTeilBearbeiten:		BOOL;
	nAufnahmeNr:			INT;
	
	bBtnHandZyklus:			BOOL;
END_VAR

//********************************************************************************
//Schrittbetrieb
fbSchrittbetrieb(	eAblaufStatus := eAblaufStatus,
					stStationInfo := stStationInfo,
					bRstInPos := bRstInPos,
					bAblaufAktiv := fbSchrittbetrieb.bAblaufAktiv OR bTeilBearbeiten);
					
fbSchrittbetrieb.bAblaufAktiv := FALSE;

//********************************************************************************					
//Handzyklus
//IF			bBtnHandZyklus THEN
//	bBtnHandZyklus := FALSE;
//	
//	IF			stStationInfo.bZyklusFertig
//		AND		bRstInPos
//		AND NOT MAIN.bProduzieren THEN
//		IF			MAIN.hatAufnBeiStJob(stStationInfo.nStationsNr) THEN							//Aufnahme will bearbeitet werden (Teile wurden schon bestellt)
//			ifStation.bearbeitenAnfordern(MAIN.getAufnahmeBeiStation(stStationInfo.nStationsNr));	//Aktuelle Aufnahme wird verwendet
//		ELSE																						//Aufnahme will NICHT bearbeitet werden (Teile müssen bestellt werden)
//			MAIN.vorwahlPseudoaufnahme();
//			ifStation.bearbeitenAnfordern(Parameter.cAnzAufnahmen+1);								//Pseudoaufnahme wird verwendet
//		END_IF	
//	END_IF
//END_IF

//********************************************************************************					
//Init
IF			stStationInfo.bInit
	AND NOT stStationInfo.bReset THEN
	stStationInfo.bInit := NOT ifStation.init();
END_IF

//********************************************************************************
//Reset
IF			bBtnReset THEN
	bBtnReset := FALSE;
	extReset();
END_IF

IF			stStationInfo.bReset THEN
	stStationInfo.bReset := NOT ifStation.reset();
END_IF

IF		NOT MAIN.bE_NotHalt THEN
	eResetStatus := ResetStatus.bereit;
END_IF

//********************************************************************************					
//Ablauf
IF			stStationInfo.bInitBeendet 
	AND NOT stStationInfo.bReset
	AND NOT fbSchrittbetrieb.bInQueue THEN
	
	IF 			bTeilBearbeiten THEN
		bTeilBearbeiten := NOT ifStation.teilBearbeiten();
	END_IF
END_IF

//********************************************************************************
//Statusanzeige
IF			stStationInfo.bReset THEN
	stStationInfo.sStatus := CONCAT('reset: ', TO_STRING(eResetStatus));
ELSIF			stStationInfo.bInit THEN
	stStationInfo.sStatus := CONCAT('init: ', TO_STRING(eInitStatus));
ELSIF			stStationInfo.bInitBeendet THEN
	stStationInfo.sStatus := TO_STRING(eAblaufStatus);
ELSE
	stStationInfo.sStatus := 'default';
END_IF

METHOD bearbeitenAnfordern
VAR_INPUT
	nAufnahme:		int;
END_VAR
bTeilBearbeiten := TRUE;
nAufnahmeNr := nAufnahme;
END_METHOD

METHOD extReset
VAR_INPUT
END_VAR
eResetStatus := ResetStatus.bereit;			//Reset neu Starten bei jedem Drücken
stStationInfo.bReset := TRUE;
END_METHOD

END_FUNCTION_BLOCK

// ---- POUs/FB_Schrittbetrieb.TcPOU
FUNCTION_BLOCK FB_Schrittbetrieb
VAR_INPUT
	eAblaufStatus:			AblaufStatus;
	eHolStatus:				AblaufStatus;
	eBereitstellStatus:		AblaufStatus;
	bAblaufAktiv:			BOOL;				//Info ob ein Teil bearbetet, geholt oder bereitgestellt werden muss
	
	bAktorPosNIO:			BOOL;				//True wenn ein aktor im handbetrieb verfahren wurde
	
	stStationInfo:			REFERENCE TO ST_Station;
	bRstInPos:				BOOL;
END_VAR
VAR_OUTPUT
	bInQueue:				BOOL;				//Es wurde rueckwaerts in die Queue gefahren und die vorherige Position wurde nicht wieder erreicht
	bAblaufFreigabe:		BOOL;				//Die Aktoren im normalen Ablauf dürfen fahren (Handoverride true) (nur bis Statuswechsel true)
	bSendFalschePosError:	BOOL;				//Aktoren sollen falsche Pos senden
END_VAR
VAR
	aSchrittQueue:			ARRAY[0..Parameter.cGroesseSchrittQueue] OF ST_SchrittQueue;
	nIndex:					INT;
	i:						INT;
	
	nAktPosition:			INT;				//Aktuelle Position in Queue
	nSollAktPos:			INT;				//Welche position andgefahren werden soll (wechselt schon wenn bewegung ausgefuehrt aber Sensoren nicht angeben)
	
	
	ePrevAblaufStatus:		AblaufStatus;
	ePrevHolStatus:			AblaufStatus;	
	ePrevBereitstellStatus:	AblaufStatus;
	
	bBtnSchrittVor:			BOOL;
	bBtnSchrittZurueck:		BOOL;
	
	bSchrittVor:			BOOL;
	bSchrittZurueck:		BOOL;
	bVorBisEnde:			BOOL;
	
	fbSendErrorTrig:		R_TRIG;
END_VAR

//********************************************************************************
//Statuswechsel erkennen
IF			ePrevAblaufStatus <> eAblaufStatus
	OR		ePrevHolStatus <> eHolStatus
	OR		ePrevBereitstellStatus <> eBereitstellStatus THEN
	
	IF			nIndex > 0 THEN
		aSchrittQueue[nIndex-1].bStatuswechsel := TRUE;
	END_IF
	
	bAblaufFreigabe := FALSE;
	
	ePrevAblaufStatus		:= eAblaufStatus;
	ePrevHolStatus			:= eHolStatus;
	ePrevBereitstellStatus	:= eBereitstellStatus;
END_IF

//********************************************************************************
//Handheld
IF			MAIN.fbHandheld.nGewaehlteStation = stStationInfo.nStationsNr THEN
	
	IF			MAIN.bE_Handbetrieb THEN
		
		IF			MAIN.fbHandheld.fbVorTrig.Q THEN
			bBtnSchrittVor := TRUE;
		ELSIF		MAIN.fbHandheld.fbZurueckTrig.Q THEN
			bBtnSchrittZurueck := TRUE;
		END_IF
		
	END_IF
END_IF

//********************************************************************************
//Zurueck zu Start wenn Anlage weiterlaeuft
IF			MAIN.bProduzieren
	AND NOT MAIN.bE_Handbetrieb
	AND		bInQueue
	AND NOT bSchrittZurueck
	AND NOT bSchrittVor THEN
	bVorBisEnde := TRUE;
	bBtnSchrittVor := TRUE;
ELSIF		MAIN.bE_Handbetrieb
	OR	NOT bInQueue THEN
	bVorBisEnde := FALSE;
END_IF

//********************************************************************************
//Aktoren fehler senden lassen wenn pos NIO 
fbSendErrorTrig(CLK := 			bAktorPosNIO 
						AND		(bBtnSchrittVor 
						OR 		bBtnSchrittZurueck),
				Q => bSendFalschePosError);

//********************************************************************************
//Schrittausloesung
IF 		NOT MAIN.bE_Handbetrieb THEN		//Zurück geht nur im Handbetrieb (vor geht auch wenn bis zum Ende gefahren weden mus)
	bBtnSchrittZurueck := FALSE;
END_IF

IF			(MAIN.bE_Handbetrieb
	OR		bVorBisEnde)
	AND	NOT bAktorPosNIO THEN
	
	IF			bBtnSchrittVor THEN
		bBtnSchrittVor := FALSE;
		
		IF			bSchrittZurueck THEN
			bSchrittZurueck := FALSE;
			nAktPosition := nSollAktPos;
		END_IF
	
		bSchrittVor := TRUE;			//Kann nur gesetzt werden wenn bSchrittZueuck nicht gesetzt ist
	END_IF
	
	IF			bBtnSchrittZurueck THEN
		bBtnSchrittZurueck := FALSE;
		
		//Wenn ein Schritt im Ablauf nicht fertig wird kann trozdem zurueck gefahren werden
		IF			bAblaufFreigabe THEN
			bAblaufFreigabe := FALSE;
		END_IF
		
		IF			bSchrittVor THEN
			bSchrittVor := FALSE;
			nAktPosition := nSollAktPos;
		END_IF
		
		bSchrittZurueck := TRUE;			//Kann nur gesetzt werden wenn bSchrittZueuck nicht gesetzt ist
	END_IF
ELSE
	bBtnSchrittVor := FALSE;
	bBtnSchrittZurueck := FALSE;
	bAblaufFreigabe := FALSE;
END_IF

//********************************************************************************
//Aktor Pos NIO reset damit die aktoren erneut setzen koennen im naechsten zuecklus
bAktorPosNIO := FALSE;

//********************************************************************************
//Schrittauslösung Ausführen
IF			bSchrittVor THEN
	bSchrittVor := NOT schrittVor();
END_IF

IF			bSchrittZurueck THEN
	bSchrittZurueck := NOT schrittZurueck();
END_IF

METHOD addToQueue
VAR_INPUT
	stEintrag:			ST_SchrittQueue;
END_VAR
VAR
	i:					INT;
END_VAR
//Bewegungen nicht aufnehmen wenn in der Queue verfahren wird
IF			bInQueue
	OR		bSchrittVor
	OR		bSchrittZurueck THEN
	RETURN;
END_IF


IF			(nIndex > Parameter.cGroesseSchrittQueue) THEN
	nIndex := Parameter.cGroesseSchrittQueue;
	
	//Alle Eintraege schieben, aelteste faellt raus
	FOR i:=1 TO Parameter.cGroesseSchrittQueue DO
		aSchrittQueue[i-1] := aSchrittQueue[i];
	END_FOR
END_IF

//In Queue aufnehmen und Message zurueckgeben
aSchrittQueue[nIndex] := stEintrag;
nAktPosition := nIndex;
nIndex := nIndex+1;
END_METHOD

METHOD reset
VAR_INPUT
END_VAR
VAR
	i:						INT;
	stTempLeer:				ST_SchrittQueue;
END_VAR
//Alle Eintraege schieben, aelteste faellt raus
FOR i:=0 TO Parameter.cGroesseSchrittQueue DO
	aSchrittQueue[i] := stTempLeer;
END_FOR
nIndex 			:= 0;
nAktPosition 	:= 0;
bInQueue 		:= FALSE;
bSchrittVor 	:= FALSE;
bSchrittZurueck := FALSE;
bAblaufFreigabe := FALSE;
END_METHOD

METHOD PRIVATE schrittVor : BOOL
VAR_INPUT
END_VAR
VAR
	i:						INT;
	nIndexbStatuswechsel:	INT;
	bPosErreicht: 			BOOL;
END_VAR
IF		NOT bRstInPos THEN
	RETURN;
END_IF

//return wenn Ende erreicht
IF			nAktPosition >= (nIndex-1) THEN
	bAblaufFreigabe := bAblaufAktiv;
	bInQueue := FALSE;
	schrittVor := TRUE;
	RETURN;
END_IF

//********************************************************************************
FOR i:= nAktPosition+1 TO nIndex-1 DO	
	nIndexbStatuswechsel := i;
	nSollAktPos := i;					//Ist immer aktuell wenn for verlassen wird
	
	IF 			aSchrittQueue[i].bGesetzt THEN			
		//*****************************************************************
		IF			__ISVALIDREF(aSchrittQueue[i].fbAktor) THEN
			aSchrittQueue[i].fbAktor.bHandOverride := TRUE;
			aSchrittQueue[i].bInPos := aSchrittQueue[i].fbAktor.arbeitsPos();
			aSchrittQueue[i].fbAktor.bHandOverride := FALSE;
		ELSIF		__ISVALIDREF(aSchrittQueue[i].fbOutput) THEN
			aSchrittQueue[i].fbOutput.bHandOverride := TRUE;
			aSchrittQueue[i].bInPos := aSchrittQueue[i].fbOutput.set();
			aSchrittQueue[i].fbOutput.bHandOverride := FALSE;
		ELSE
			//Fehler!!!
			i := i-1;
			EXIT;
		END_IF
		//*****************************************************************
	ELSE
		//*****************************************************************
		IF			__ISVALIDREF(aSchrittQueue[i].fbAktor) THEN
			aSchrittQueue[i].fbAktor.bHandOverride := TRUE;
			aSchrittQueue[i].bInPos := aSchrittQueue[i].fbAktor.ruhePos();
			aSchrittQueue[i].fbAktor.bHandOverride := FALSE;
		ELSIF		__ISVALIDREF(aSchrittQueue[i].fbOutput) THEN
			aSchrittQueue[i].fbOutput.bHandOverride := TRUE;
			aSchrittQueue[i].bInPos := aSchrittQueue[i].fbOutput.reset();
			aSchrittQueue[i].fbOutput.bHandOverride := FALSE;
		ELSE
			//Fehler!!!
			i := i-1;
			EXIT;
		END_IF
		//*****************************************************************
	END_IF
	
	IF		aSchrittQueue[i].bStatuswechsel THEN
		EXIT;
	END_IF
END_FOR

//********************************************************************************
bPosErreicht := TRUE;
FOR i:= nAktPosition+1 TO nIndexbStatuswechsel DO
	IF		NOT	aSchrittQueue[i].bInPos THEN
		bPosErreicht := FALSE;
	END_IF
END_FOR

//Alle inPos bei jedem Aufruf zuruecksetzten
FOR i:= nAktPosition+1 TO nIndexbStatuswechsel DO
	aSchrittQueue[i].bInPos := FALSE;
END_FOR

IF			bPosErreicht THEN
	nAktPosition := nIndexbStatuswechsel;
	IF			nAktPosition = (nIndex-1) THEN
		bInQueue := FALSE;
	END_IF	
	schrittVor := TRUE;	
END_IF
END_METHOD

METHOD PRIVATE schrittZurueck : BOOL
VAR_INPUT
END_VAR
VAR
	i:						INT;
	nIndexbStatuswechsel:	INT;
	bPosErreicht: 			BOOL;
	
	nPosVorher:				INT;
END_VAR
IF		NOT bRstInPos THEN
	RETURN;
END_IF

IF			nAktPosition >= 0 THEN
	bInQueue := TRUE;
ELSE									//Wenn noch kein Schritt aufgezeichnet wurde -> return True
	schrittZurueck := TRUE;
	RETURN;
END_IF

//********************************************************************************
FOR i:= nAktPosition TO 0 BY -1 DO
	nIndexbStatuswechsel := i;
	nSollAktPos := i;					//Ist immer aktuell wenn for verlassen wird

	IF		NOT aSchrittQueue[i].bStatuswechsel
		OR		i = nAktPosition THEN
			
		IF 			aSchrittQueue[i].bGesetzt THEN			
			//*****************************************************************
			IF			__ISVALIDREF(aSchrittQueue[i].fbAktor) THEN
				aSchrittQueue[i].fbAktor.bHandOverride := TRUE;
				aSchrittQueue[i].bInPos := aSchrittQueue[i].fbAktor.ruhePos();
				aSchrittQueue[i].fbAktor.bHandOverride := FALSE;
			ELSIF		__ISVALIDREF(aSchrittQueue[i].fbOutput) THEN
				aSchrittQueue[i].fbOutput.bHandOverride := TRUE;
				aSchrittQueue[i].bInPos := aSchrittQueue[i].fbOutput.reset();
				aSchrittQueue[i].fbOutput.bHandOverride := FALSE;
			ELSE
				//Fehler!!!
				EXIT;
			END_IF
			//*****************************************************************
		ELSE
			//*****************************************************************
			IF			__ISVALIDREF(aSchrittQueue[i].fbAktor) THEN
				aSchrittQueue[i].fbAktor.bHandOverride := TRUE;
				aSchrittQueue[i].bInPos := aSchrittQueue[i].fbAktor.arbeitsPos();
				aSchrittQueue[i].fbAktor.bHandOverride := FALSE;
			ELSIF		__ISVALIDREF(aSchrittQueue[i].fbOutput) THEN
				aSchrittQueue[i].fbOutput.bHandOverride := TRUE;
				aSchrittQueue[i].bInPos := aSchrittQueue[i].fbOutput.set();
				aSchrittQueue[i].fbOutput.bHandOverride := FALSE;
			ELSE
				//Fehler!!!
				EXIT;
			END_IF
			//*****************************************************************
		END_IF
		
		//Wenn i=0 ist und der Schritt in Queue[0] ausgeführt wurde muss index -1 sein damit Queue[0] beim vorwärts fahren wieder ausgeführt wird
		IF			i = 0 THEN
			nIndexbStatuswechsel := -1;
			nSollAktPos := -1;
		END_IF
		
	ELSIF		aSchrittQueue[i].bStatuswechsel
		AND		i <> nAktPosition THEN
		EXIT;
	END_IF
END_FOR

//********************************************************************************
//Abfrage alle in Pos
bPosErreicht := TRUE;
FOR i:= nAktPosition TO nIndexbStatuswechsel+1 BY -1 DO
	IF		NOT	aSchrittQueue[i].bInPos THEN
		bPosErreicht := FALSE;
	END_IF
END_FOR

//Alle inPos bei jedem Aufruf zuruecksetzten
FOR i:= nAktPosition TO nIndexbStatuswechsel+1 BY -1 DO
	aSchrittQueue[i].bInPos := FALSE;
END_FOR

IF			bPosErreicht THEN
	nAktPosition := nIndexbStatuswechsel;
	schrittZurueck := TRUE;
END_IF
END_METHOD

METHOD vor
VAR_INPUT
END_VAR
bBtnSchrittVor := TRUE;
END_METHOD

METHOD zurueck
VAR_INPUT
END_VAR
bBtnSchrittZurueck := TRUE;
END_METHOD

END_FUNCTION_BLOCK

// ---- POUs/FB_Aktor.TcPOU
FUNCTION_BLOCK FB_Aktor
VAR_INPUT	
	bHandOverride:				BOOL;			//Wenn true kann der Ausgang auch im Handbetrieb geschrieben werden	
	fbSchrittbetrieb:			REFERENCE TO FB_Schrittbetrieb;
	
	//Inputs
	bE_sensRP					AT%I*:BOOL;		//VAR_INPUT damit zwischenpositionen abgefragt werden können
	bE_sensAP					AT%I*:BOOL;
	
	b53WegeVentil:				BOOL;
	
	bSensAPVorhanden:			BOOL;
	bSensRPVorhanden:			BOOL;
	tZeitAP:					TIME;
	tZeitRP:					TIME;
END_VAR
VAR_OUTPUT
	bStoerung:					BOOL;
	bFalschePos:				BOOL;
END_VAR
VAR	
	//Outputs
	bArbeitsPos:				BOOL;
	bA_arbeitsPos				AT%Q*:BOOL;	
	
	bBtnHandausloesung:			BOOL;
	
	fbZeitRP:					TON;
	fbZeitAP:					TON;
	
	eStatus:					AktorStatus;
	
	bStartUberpruefung:			BOOL;
	
	eAnfrage:					AktorStatus;
	
	fbFtrigHandbetr:			F_TRIG;
	
	
	//Parameter
	//bSensAPVorhanden:			BOOL;
	//bSensRPVorhanden:			BOOL;
	
	//tZeitRP:					TIME := T#2S;
	//tZeitAP:					TIME := T#2S;
	
	bStoerungRP: 				BOOL;
	bStoerungAP: 				BOOL;

	
	nErrorIdAP:					INT;
	nErrorIdRP:					INT;
	
	sBezeichnung:				STRING;			//Bezeichnung für Handbetriebfehlermeldung
END_VAR

bA_arbeitsPos := bArbeitsPos AND (NOT MAIN.bE_SafetyProgStop AND MAIN.bE_LuftdruckIO OR NOT b53WegeVentil);

fbZeitAP(PT:=tZeitAP, IN := 			bA_arbeitsPos
								AND (NOT bSensAPVorhanden
								OR	NOT bE_sensAP
								OR		bSensRPVorhanden
								AND 	bE_sensRP));

fbZeitRP(PT:=tZeitRP, IN := 		NOT bA_arbeitsPos
								AND (NOT bSensRPVorhanden
								OR NOT	bE_sensRP
								OR		bSensAPVorhanden
								AND		bE_sensAP));

//Fehlermeldungen
IF			bSensAPVorhanden
	AND		fbZeitAP.Q 
	AND		bStartUberpruefung
	AND NOT bStoerungAP
	AND NOT (nErrorIdAP = 0) THEN

	EventLogger.aAlarm[nErrorIdAP].Raise(0);
	bStoerungAP := TRUE;

ELSIF		NOT	fbZeitAP.Q 
		AND		bStoerungAP THEN
	EventLogger.aAlarm[nErrorIdAP].Clear(0, TRUE);
	bStoerungAP := FALSE;
END_IF

IF			bSensRPVorhanden
	AND		fbZeitRP.Q 
	AND		bStartUberpruefung
	AND NOT bStoerungRP
	AND NOT (nErrorIdRP = 0) THEN
	
	EventLogger.aAlarm[nErrorIdRP].Raise(0);
	bStoerungRP := TRUE;
	
ELSIF		NOT fbZeitRP.Q
		AND		bStoerungRP THEN
		
	EventLogger.aAlarm[nErrorIdRP].Clear(0, TRUE);
	bStoerungRP := FALSE;
END_IF

bStoerung := bStoerungAP OR bStoerungRP;

//Status
//http://www.32x8.com/sop6_____A-B-C-D-E-F_____m_33-35-37-39-41-45-52-53-54-55-60-61___________option-0_____989781876978894288722
IF			bA_arbeitsPos
			AND	(NOT bSensAPVorhanden
			AND	NOT bSensRPVorhanden
			AND		fbZeitAP.Q
			
